// POUs/Motion/TF511x-KIN/03_DUTs/Trafo/KIN_STATICTRAFO_PARAM
{attribute 'hide'}
FUNCTION_BLOCK KIN_STATICTRAFO_PARAM
VAR_INPUT
	oid														:	UDINT := 0;
	TranslationX											:	LREAL := 0.0;
	TranslationY											:	LREAL := 0.0;
	TranslationZ											:	LREAL := 0.0;
                            								
	Rotation												: LREAL := 0.0;
	RotationAxis											: INT := 2;

END_VAR
VAR_OUTPUT

END_VAR
VAR
END_VAR

;

METHOD delete : BOOL
VAR_INPUT
END_VAR
	oid														:= 0;
	TranslationX											:= 0.0;
	TranslationY											:= 0.0;
	TranslationZ											:= 0.0;
                            								
	Rotation												:= 0.0;
	RotationAxis											:= 2;
delete	:= TRUE;
END_METHOD

END_FUNCTION_BLOCK

// POUs/Motion/TF511x-KIN/03_DUTs/Trafo/KIN_TOOLTRAFO_PARAM
{attribute 'hide'}
FUNCTION_BLOCK KIN_TOOLTRAFO_PARAM
VAR_INPUT
	oid														:	UDINT := 0;
	dx														: 	LREAL := 0.0;  (* Default Tooldata at WOS *)
	dy														: 	LREAL := 0.0;  (* Default Tooldata at WOS *)
	dz														:	LREAL := 0.0;  (* Default Tooldata at WOS *)

END_VAR
VAR_OUTPUT

END_VAR
VAR
END_VAR

;

METHOD delete : BOOL
VAR_INPUT
END_VAR
	oid														:= 0;
	dx														:= 0.0;  (* Default Tooldata at WOS *)
	dy														:= 0.0;  (* Default Tooldata at WOS *)
	dz														:= 0.0;  (* Default Tooldata at WOS *)
delete	:= TRUE;
END_METHOD

END_FUNCTION_BLOCK

// POUs/Motion/TF511x-KIN/KinChannel
FUNCTION_BLOCK KinChannel EXTENDS KIN_REF
VAR_INPUT
	Admin													:	KinAdmin;
END_VAR
VAR_OUTPUT
END_VAR
VAR
END_VAR

(* Kinematic Ctrl 										*)
(********************************************************)

(* work IO ********************************************************************)
(*	IO(); *)
	
(****************************************************************************)
(* Kinematic group control													*)
(****************************************************************************)
	Admin(
		ResetTrig			:= ,
		Enable			:= ,
		Override		:= ,
		ItpChannelId	:= ,
		AxesList		:= ,
		rKINRef			:= THIS^,
		Busy			=> ,
		Done			=> ,
		Error			=> ,
		ErrorId			=> );
(****************************************************************************)

END_FUNCTION_BLOCK

// POUs/Motion/VALUE_3D
{attribute 'no_check'}
FUNCTION_BLOCK VALUE_3D
VAR_INPUT                                                            
	Valid													:	BOOL ;
	X														:	LREAL;
	Y														:	LREAL;
	Z														:	LREAL;
END_VAR
VAR_OUTPUT
END_VAR
VAR
END_VAR

;

METHOD PUBLIC copy : BOOL //Return value = TRUE if execution finished
VAR_IN_OUT
	Source													:	VALUE_3D;
END_VAR
	Valid													:= Source.Valid;
	X														:= Source.X;
	Y														:= Source.Y;
	Z														:= Source.Z;
	copy													:= TRUE;
END_METHOD

METHOD PUBLIC delete : BOOL //Return value = TRUE if execution finished - Valid bit will not change
VAR_INPUT
END_VAR
	X					 									:= 0.0;	
	Y					 									:= 0.0;	
	Z					 									:= 0.0;	
	delete													:= TRUE;
END_METHOD

METHOD PUBLIC InPos : BOOL //Return value = TRUE axes is within window of checkPos values
VAR_IN_OUT
	CheckPos												:	VALUE_3D;
	Window													:	VALUE_3D;
END_VAR
InPos														:= CAM(CheckPos.X, X ,Window.X)
																AND CAM(CheckPos.Y, Y ,Window.Y)
																AND CAM(CheckPos.Z, Z ,Window.Z);
END_METHOD

METHOD PUBLIC InPosByAxisNo : BOOL //Return value = TRUE selected axis is within window of checkPos values
VAR_INPUT
	No					:	INT;
END_VAR
VAR_IN_OUT
	CheckPos			:	VALUE_3D;
	Window				:	VALUE_3D;
END_VAR
InPosByAxisNo													:= (CAM(CheckPos.X, X ,Window.X) OR No <> 1)
																AND (CAM(CheckPos.Y, Y ,Window.Y) OR No <> 2)
																AND (CAM(CheckPos.Z, Z ,Window.Z) OR No <> 3);
END_METHOD

METHOD PUBLIC InPosXY : BOOL //Return value = TRUE if axes are within window of checkPos values
VAR_IN_OUT
	CheckPos			:	VALUE_3D;
	Window				:	VALUE_3D;
END_VAR
InPosXY 													:= CAM(CheckPos.X, X ,Window.X)
																AND CAM(CheckPos.Y, Y ,Window.Y);
END_METHOD

METHOD PUBLIC InPosXZ : BOOL //Return value = TRUE if axes are within window of checkPos values
VAR_IN_OUT
	CheckPos			:	VALUE_3D;
	Window				:	VALUE_3D;
	
END_VAR
InPosXZ														:= CAM(CheckPos.X, X ,Window.X)
																AND CAM(CheckPos.Z, Z ,Window.Z);
END_METHOD

METHOD PUBLIC InPosYZ : BOOL //Return value = TRUE if axes are within window of checkPos values
VAR_IN_OUT
	CheckPos			:	VALUE_3D;
	Window				:	VALUE_3D;
	
END_VAR
InPosYZ													:= CAM(CheckPos.Y, Y ,Window.Y)
																AND CAM(CheckPos.Z, Z ,Window.Z);
END_METHOD

METHOD PUBLIC reset : BOOL //Delete data and reset valid , TRUE if execution finished
VAR_INPUT
END_VAR
Delete();
Valid														:= FALSE;
reset														:= TRUE;
END_METHOD

END_FUNCTION_BLOCK

// POUs/Motion/VALUE_6D
{attribute 'no_check'}
FUNCTION_BLOCK VALUE_6D 
VAR_INPUT
	Valid													:	BOOL ;
	X														:	LREAL;
	Y														:	LREAL;
	Z														:	LREAL;
	A														:		LREAL; //Rx
	B														:		LREAL; //Ry
	C														:		LREAL; //Rz	
END_VAR
VAR_OUTPUT
END_VAR
VAR
END_VAR

;

METHOD PUBLIC copy : BOOL //Return value = TRUE if execution finished
VAR_IN_OUT
	Source													:	VALUE_6D;
END_VAR
	Valid													:= Source.Valid;
	X														:= Source.X;
	Y														:= Source.Y;
	Z														:= Source.Z;
	A														:= Source.A;
	B														:= Source.B;
	C														:= Source.C;
	copy													:= TRUE;
END_METHOD

METHOD PUBLIC delete : BOOL //Return value = TRUE if execution finished - Valid bit will not change
VAR_INPUT
END_VAR
	X					 									:= 0.0;	
	Y					 									:= 0.0;	
	Z					 									:= 0.0;	
	A						 								:= 0.0;	
	B						 								:= 0.0;	
	C						 								:= 0.0;	
	delete													:= TRUE;
END_METHOD

METHOD PUBLIC inPos : BOOL //Return value = TRUE if axes are within window of checkPos values
VAR_IN_OUT
	CheckPos												:	VALUE_6D;
	Window													:	VALUE_6D;
END_VAR             										
VAR CONSTANT        										
END_VAR
InPos 														:= CAM(CheckPos.X, X, Window.X)
																AND CAM(CheckPos.Y, Y ,Window.Y)
																AND CAM(CheckPos.Z, Z,Window.Z)
																AND CAM(CheckPos.A, A, Window.A)
																AND CAM(CheckPos.B, B ,Window.B)
																AND CAM(CheckPos.C, C,Window.C);
END_METHOD

METHOD PUBLIC InPosABC : BOOL //Return value = TRUE if axes are within window of checkPos values
VAR_IN_OUT
	CheckPos												:	VALUE_6D;
	Window													:	VALUE_6D;
END_VAR                 									
VAR CONSTANT            									
END_VAR
InPosABC												 	:= CAM(CheckPos.A, A ,Window.A)
																AND CAM(CheckPos.B, B ,Window.B)
																AND CAM(CheckPos.C, C ,Window.C);
END_METHOD

METHOD PUBLIC InPosAC : BOOL //Return value = TRUE if axes are within window of checkPos values
VAR_IN_OUT
	CheckPos												:	VALUE_6D;
	Window													:	VALUE_6D;
END_VAR                 									
VAR CONSTANT            									
END_VAR
InPosAC													 	:= CAM(CheckPos.A, A ,Window.A)
																AND CAM(CheckPos.C, C ,Window.C);
END_METHOD

METHOD PUBLIC inPosByAxisNo : BOOL //Return value = TRUE selected axis is within window of checkPos values
VAR_INPUT
	No					:	INT;
END_VAR
VAR_IN_OUT
	CheckPos			:	VALUE_6D;
	Window				:	VALUE_6D;
END_VAR
inPosByAxisNo													:= (CAM(CheckPos.X, X ,Window.X) OR No <> 1)
																AND (CAM(CheckPos.Y, Y ,Window.Y) OR No <> 2)
																AND (CAM(CheckPos.Z, Z ,Window.Z) OR No <> 3)
																AND (CAM(CheckPos.A, A ,Window.A) OR No <> 4)
																AND (CAM(CheckPos.B, B ,Window.B) OR No <> 5)
																AND (CAM(CheckPos.C, C ,Window.C) OR No <> 6);
END_METHOD

METHOD PUBLIC inPosXY : BOOL //Return value = TRUE if axes are within window of checkPos values
VAR_IN_OUT
	CheckPos												:	VALUE_6D;
	Window													:	VALUE_6D;
END_VAR                 									
VAR CONSTANT            									
END_VAR
InPosXY													 	:= CAM(CheckPos.X, X ,Window.X)
																AND CAM(CheckPos.Y, Y ,Window.Y);
END_METHOD

METHOD PUBLIC InPosXYZ : BOOL //Return value = TRUE if axes are within window of checkPos values
VAR_IN_OUT
	CheckPos												:	VALUE_6D;
	Window													:	VALUE_6D;
END_VAR                 									
VAR CONSTANT            									
END_VAR
InPosXYZ												 	:= CAM(CheckPos.X, X ,Window.X)
																AND CAM(CheckPos.Y, Y ,Window.Y)
																AND CAM(CheckPos.Z, Z ,Window.Z);
END_METHOD

METHOD PUBLIC inPosXZ : BOOL //Return value = TRUE if axes are within window of checkPos values
VAR_IN_OUT
	CheckPos												:	VALUE_6D;
	Window													:	VALUE_6D;
END_VAR                 									
VAR CONSTANT            									
END_VAR
InPosXZ												 	:= CAM(CheckPos.X, X ,Window.X)
																AND CAM(CheckPos.Z, Z ,Window.Z);
END_METHOD

METHOD PUBLIC inPosYZ : BOOL //Return value = TRUE if axes are within window of checkPos values
VAR_IN_OUT
	CheckPos												:	VALUE_6D;
	Window													:	VALUE_6D;
END_VAR                 									
VAR CONSTANT            									
END_VAR
InPosYZ													 	:= CAM(CheckPos.Y, Y ,Window.Y)
																AND CAM(CheckPos.Z, Z ,Window.Z);
END_METHOD

METHOD PUBLIC reset : BOOL //Delete data and reset valid , TRUE if execution finished
VAR_INPUT
END_VAR
Delete(); 
Valid														:= FALSE;
reset														:= TRUE;
END_METHOD

END_FUNCTION_BLOCK

// POUs/Safety/Diag/SafetyIODeviceDiag_wEvents
{attribute 'no_check'}
FUNCTION_BLOCK SafetyIODeviceDiag_wEvents
VAR CONSTANT
	MIN_EVENT												:	INT := 1;
	MAX_EVENT												:	INT := 10;
	
//Event conn diag code xxxx					| FB1 - Msg 1..15
//Event conn diag code .4 					| FB2 - Msg 16
//Event conn diag code .5 					| FB3 - Msg 17
                                        	
//Event internal error 						| FB1 - Msg 18
                                        	
//Event send TextId 						| FB4 - Msg 19
                                        	
//Event send AX5xxx Err Chn 1 				| FB5 - Msg 20
//Event send AX5xxx Err Chn 1 				| FB6 - Msg 21
                                        	
//Event send Ex19 Err Debug 0x800E:0A 		| FB4 - Msg 22
//Event send Ex19 Err Debug 0x800E:0B		| FB5 - Msg 23
//Event send Ex19 Err Debug 0x800E:0C 		| FB6 - Msg 24
//Event send Ex19 Err Debug 0x800E:0D 		| FB7 - Msg 25
//Event send Ex19 Err Debug 0x800E:13 		| FB8 - Msg 26
//Event send Ex19 Err Debug 0x800E:14 		| FB9 - Msg 27
//Event send Ex19 Err Debug 0x800E:15		| FB10- Msg 28
                                        	
//Event send EL29 Err Debug 0x800E:0C 		| FB4 - Msg 30 (Querschluss bit 0..3)
//Event send EL29 Err Debug 0x800E:0C 		| FB4 - Msg 31 (Open load bit 4..7)
//Event send EL29 Err Debug 0x800E:0D		| FB5 - Msg 32
//Event send EL29 Err Debug 0x800E:0E 		| FB6 - Msg 33
//Event send EL29 Err Debug 0x800E:0E 		| FB7 - Msg 34
//Event send EL29 Err Debug 0x800E:0E 		| FB8 - Msg 35

                                        	
//Event send EK19 Err Debug 0x800E:0A		| FB4 - Msg 22 
//Event send EK19 Err Debug 0x800E:0B		| FB5 - Msg 23 
//Event send EK19 Err Debug 0x800E:0C 		| FB6 - Msg 24 
//Event send EK19 Err Debug 0x800E:0D 		| FB7 - Msg 25 
//Event send EK19 Err Debug 0x800E:0E	 	| FB8 - Msg 36..45
END_VAR
VAR_INPUT
	Enable													:	BOOL;	//FB will be processed as long as enable is TRUE 
	ConfirmTrig												:	BOOL;	//Resets error with rising edge 
	SourceId												:	UDINT;	//Multisource id 
	EcMasterDevId											:	UINT;	//Map to EtherCAT Master DevId
END_VAR                 									
VAR_OUTPUT              									
	Connected												:	BOOL;
	{attribute 'displaymode':='binary'}
	Status													:	DWORD;	//current status of event
	NoOfActiveEvents										:	INT;
END_VAR                 									

VAR(* internal *)
	state													:	INT := 0;
	{attribute 'displaymode':='binary'}
	ConnMsgDiagCode											:	BYTE;
	Read													:	SafetyIODeviceDiagRead;
   	Event													:	ARRAY [MIN_EVENT..MAX_EVENT] OF EventHandling; 
	DevTypeAndAddr											:	STRING(30);
    DebugData												:	 word;                 								                            	
	i														:	INT;
END_VAR

(* Safety IO device diag with events		V2	*)
(************************************************)

(* Status connected ***************************************************)
	Connected 												:= Read.AdsAddr.port <> 0;
	
(* Read adress and type ***********************************************)
	IF Enable AND Connected AND Read.MsgInfoDiag <> 0 OR State <> 0
	THEN
		CASE State OF
		0:	
			IF Read.MsgInfoDiag <> 0
			THEN
				Read(Execute := FALSE);
				Read(Execute := TRUE, EcMasterDevId := EcMasterDevId);
				State										:= State + 1;
			END_IF
			
		1: //Read diag data from device
			Read(Execute := TRUE, EcMasterDevId := EcMasterDevId);
			IF NOT Read.Busy
			THEN
	
				IF Read.Error
				THEN
					Event[1].Text1							:= SEL(Read.Name = '',Read.Name , '<ERR_READ_DIAG>');
					DevTypeAndAddr							:= SEL(Read.DevType = '', Read.DevType, '<Unknown>');
					DevTypeAndAddr							:= CONCAT(DevTypeAndAddr, CONCAT(' (Ec Addr.', CONCAT(TO_STRING(Read.AdsAddr.port),')')));	
					Event[1].Text2							:= CONCAT(' - ErrorID ', DWORD_TO_HEXSTR(TO_DWORD(Read.ErrorID),4,FALSE));
					Event[1].Text2							:= CONCAT(Event[1].Text2 , CONCAT(' in state ', TO_STRING(Read.DiagMsgTextId)));
					Event[1].SourceId						:= SourceId;
					Event[1].Flag							:= TRUE;
					State									:= 98;
				ELSIF Event[1].SourceId = 0
				THEN //Init device information 
					FOR i := MIN_EVENT TO MAX_EVENT
					DO
						Event[i].Text1						:= Read.Name;
						DevTypeAndAddr						:= CONCAT(Read.DevType, ' (FSOE Addr.');
						DevTypeAndAddr						:= CONCAT(DevTypeAndAddr, CONCAT(TO_STRING(Read.FSOEAddr), ')'));	
						Event[i].SourceId					:= SourceId;
					END_FOR
					State									:= 99;
				ELSE
					State									:= 99;
				END_IF		
				Read(Execute := FALSE);
			END_IF
			
		98: //Show internal error
			Event[1](
				Flag	:= Event[1].Flag AND NOT Event[1].ConfirmTrig,
				ConfirmTrig:= ConfirmTrig OR Read.MsgInfoDiag = 0, 
				MsgId	:= 18, 
				pText3	:= ADR(DevTypeAndAddr),
				Status	=> Status);	
			IF NOT Event[1].Status.31 
			THEN
				NoOfActiveEvents							:= 0;
				state										:= 0;
			ELSE
				NoOfActiveEvents							:= 1;
			END_IF
			
		99: //Fire events
			IF Read.MsgInfoDiag = 0 AND NOT Status.31
			THEN //Go back to 0 if messages cleared
				State 										:= 0;
			ELSE
				//Show connection error events
				_eventsConnDiag();
				
				//Fire device events
				IF Read.pDebugData <> 0 
				THEN //Safety devices without diag history object
					IF Read.DebugDataMaxId = 16#08 AND_THEN FIND(Read.DevType, 'AX580') <> 0
					THEN
						_eventsAX580x(Read.MsgInfoDiag <> 0);
					ELSIF Read.DebugDataMaxId = 16#10 AND_THEN Read.DevType = 'EL2904'
					THEN
						_eventsEL2904(Read.MsgInfoDiag <> 0);
					ELSIF Read.DebugDataMaxId = 16#40 AND_THEN Read.DevType = 'EK1914' 
					THEN
						_eventsEK1914(Read.MsgInfoDiag <> 0);
					ELSIF Read.DebugDataMaxId >= 16#10 
					THEN//EL1904 or EP1908
						_eventsEx190x(Read.MsgInfoDiag <> 0);		
					ELSE //Show internal error 
						Event[4](
							Flag	:= Read.MsgInfoDiag <> 0,
							ConfirmTrig:= ConfirmTrig OR Read.MsgInfoDiag = 0, 
							MsgId	:= 18, 
							Text2	:= CONCAT(' Invalid lenght of Coe object 0x800E for device ', TO_STRING(Read.DebugDataMaxId)),
							pText3	:= ADR(DevTypeAndAddr));	
					END_IF
				ELSE //TwinSAFE terminal with diag history  
					_eventsDiagHistory(Read.MsgInfoDiag <> 0);
				END_IF			
			END_IF		
						   	
			//Check whether one event is active **************************************
			NoOfActiveEvents 		 						:= 0;			
			Status											:= 0;						
			FOR i := MIN_EVENT TO MAX_EVENT
			DO 
				IF Event[i].Status.31 THEN NoOfActiveEvents := NoOfActiveEvents + 1 ; END_IF
				Status										:= Status OR Event[i].Status;
			END_FOR
		END_CASE
	END_IF

(*******************************************************************************)

METHOD PRIVATE _eventsAX580x : BOOL
VAR_INPUT
	ShowEvent										:	BOOL;
END_VAR
(* Fire AX5000 events ***********************************)
	//Send AX58xx diag code channel 1 
	IF Read.pDebugData^[1] = 0
	THEN
		Event[5].Text2										:= CONCAT('0x',DWORD_TO_HEXSTR(TO_DWORD(Read.pDebugData^[7]),4,FALSE));
	ELSE
		Event[5].Text2										:= '<Set CoE object 0xFA10:01 = 0>';
	END_IF
 
	Event[5](
		Flag	:= ShowEvent AND Read.msgSevyIsError ,
		ConfirmTrig:= ConfirmTrig, 
		MsgId	:= 20, 
		Class	:= ,
		pText3	:= ADR(DevTypeAndAddr));	
		
	//Send AX58xx diag code channel 2
	IF Read.pDebugData^[1] = 0
	THEN
		Event[6].Text2										:= CONCAT('0x',DWORD_TO_HEXSTR(TO_DWORD(Read.pDebugData^[8]),4,FALSE));
	ELSE
		Event[6].Text2										:=  '<Set CoE object 0xFA10:01 = 0>';
	END_IF
 
	Event[6](
		Flag	:= ShowEvent AND Read.msgSevyIsError ,
		ConfirmTrig:= ConfirmTrig, 
		MsgId	:= 21, 
		Class	:= ,
		pText3	:= ADR(Read.Name));

(******************************************************)
END_METHOD

METHOD PRIVATE _eventsConnDiag : BOOL
VAR_INPUT
END_VAR
(* Fire event for connection error code ************************************)
	ConnMsgDiagCode											:= 16#0F AND Read.MsgInfoDiag; 
	IF ConnMsgDiagCode <> 0 OR Event[1].Status.31
	THEN
		Event[1](
			Flag	:= ConnMsgDiagCode <> 0 AND NOT (ConnMsgDiagCode = 2#1101 AND Read.MsgInfoDiag.5),
			ConfirmTrig:= ConfirmTrig, 
			MsgId	:= ConnMsgDiagCode,  //1..15 		
			pText3	:= ADR(DevTypeAndAddr));	
	END_IF
	
	//Fire event xxx1 xxxx FSoE Slave error detected
	IF Read.MsgInfoDiag.4 OR Event[2].Status.31
	THEN
		Event[2](
			Flag	:= Read.MsgInfoDiag.4,
			ConfirmTrig:= ConfirmTrig, 
			MsgId	:= 16,		
			pText3	:= ADR(DevTypeAndAddr));	
	END_IF

(*
	//Fire event xx1x xxxx FSoE Slave notifies Failsafe Value active
	IF Read.MsgInfoDiag.5 OR Event[3].Status.31
	THEN
		Event[3](
			Flag	:= Read.MsgInfoDiag.5,
			ConfirmTrig:= ConfirmTrig, 
			MsgId	:= 17,		
			pText3	:= ADR(DevTypeAndAddr));		
	END_IF
*)	
	(*
	Tabelle 2-4: Diagnose-Informationen einer Connection
	Wert Beschreibung
	xxxx 0001 invalid command
	xxxx 0010 unknown command
	xxxx 0011 invalid connection ID
	xxxx 0100 invalid CRC
	xxxx 0101 Watchdog run out of time
	xxxx 0110 invalid FSoE-Adress
	xxxx 0111 invalid data
	xxxx 1000 invalid length of communicatoin parameter Kommunikationsparameterlänge
	xxxx 1001 invalid communicatoin parameter
	xxxx 1010 invalid operator parameter length
	xxxx 1011 invalid operator parameter
	xxxx 1100 FSoE Master Reset
	xxxx 1101 Module fault on slave detected with activated option "Modulfault is ComError"
	xxxx 1110 Module fault on EL290x at activated with option "Error achnowledge active"
	xxxx 1111 Slave not started or unexpected error argument
	
	*)
		
(***********************************************************************)
END_METHOD

METHOD PRIVATE _eventsDiagHistory : BOOL
VAR_INPUT
	ShowEvent										:	BOOL;
END_VAR
(* Send diag message textId ********************************************)
	Event[4](
		Flag	:= ShowEvent AND Read.msgSevyIsError ,
		ConfirmTrig:= ConfirmTrig, 
		MsgId	:= 19, 
		Text2	:= CONCAT('0x',DWORD_TO_HEXSTR(TO_DWORD(Read.DiagMsgTextId),4,FALSE)),
		pText3	:= ADR(DevTypeAndAddr));

(******************************************************)
END_METHOD

METHOD PRIVATE _eventsEK1914 : BOOL
VAR_INPUT
	ShowEvent										:	BOOL;
END_VAR
// Fire events for of EK1914 ****************************************)

		(* error during sensor-test *)
		Event[4].Flag 										:= Read.pDebugData^[16#0A] <> 0;
		IF Event[4].Flag OR Event[4].Status.31
		THEN
			DebugData										:= Read.pDebugData^[16#0A];
			Event[4].Text2									:= '';
			IF DebugData.0 THEN Event[4].Text2 				:= CONCAT(Event[4].Text2, '|1'); END_IF
			IF DebugData.1 THEN Event[4].Text2 				:= CONCAT(Event[4].Text2, '|2'); END_IF
		(*	IF DebugData.2 THEN Event[4].Text2 				:= CONCAT(Event[4].Text2, '|3'); END_IF
			IF DebugData.3 THEN Event[4].Text2 				:= CONCAT(Event[4].Text2, '|4');  END_IF
			IF DebugData.4 THEN Event[4].Text2 				:= CONCAT(Event[4].Text2, '|5'); END_IF
			IF DebugData.5 THEN Event[4].Text2 				:= CONCAT(Event[4].Text2, '|6'); END_IF
			IF DebugData.6 THEN Event[4].Text2 				:= CONCAT(Event[4].Text2, '|7'); END_IF
			IF DebugData.7 THEN Event[4].Text2 				:= CONCAT(Event[4].Text2, '|8');  END_IF *)
			Event[4].Text2 									:= CONCAT(Event[4].Text2, '|'); 			
			
			Event[4](
				Flag	:= ShowEvent ,
				ConfirmTrig:= ConfirmTrig, 
				MsgId	:= 22, 
				pText3	:= ADR(DevTypeAndAddr))	;
		END_IF

		(* Zweikanalauswertung fehlerhaft *)
		Event[5].Flag 										:= Read.pDebugData^[16#0B] <> 0;
		IF Event[5].Flag OR Event[5].Status.31
		THEN
			DebugData										:= Read.pDebugData^[16#0B];
			Event[5].Text2									:= '';
			IF DebugData.0 THEN Event[5].Text2 				:= CONCAT(Event[5].Text2, '|1+2'); END_IF
		(*	IF DebugData.1 THEN Event[5].Text2 				:= CONCAT(Event[5].Text2, '|3+4'); END_IF
			IF DebugData.2 THEN Event[5].Text2 				:= CONCAT(Event[5].Text2, '|5+6'); END_IF
			IF DebugData.3 THEN Event[5].Text2 				:= CONCAT(Event[5].Text2, '|7+8');  END_IF *)
			Event[5].Text2 									:= CONCAT(Event[5].Text2, '|'); 
			
			Event[5](
				Flag	:= ShowEvent ,
				ConfirmTrig:= ConfirmTrig, 
				MsgId	:= 23, 
				pText3	:= ADR(DevTypeAndAddr))	;
		END_IF

		(* Fehler Eingangspaar Trittmattenbetriebsart - Eingangspaar uneinig *)
		Event[6].Flag 										:= Read.pDebugData^[16#0C] <> 0;
		IF Event[6].Flag OR Event[6].Status.31
		THEN
			DebugData										:= Read.pDebugData^[16#0C];
			Event[6].Text2									:= '';
			IF DebugData.0 THEN Event[6].Text2 				:= CONCAT(Event[6].Text2, '|1+2'); END_IF
		(*	IF DebugData.1 THEN Event[6].Text2 				:= CONCAT(Event[6].Text2, '|3+4'); END_IF
			IF DebugData.2 THEN Event[6].Text2 				:= CONCAT(Event[6].Text2, '|5+6'); END_IF
			IF DebugData.3 THEN Event[6].Text2 				:= CONCAT(Event[6].Text2, '|7+8');  END_IF *)
			Event[6].Text2 									:= CONCAT(Event[6].Text2, '|'); 
			
			Event[6](
				Flag	:= ShowEvent ,
				ConfirmTrig:= ConfirmTrig, 
				MsgId	:= 24, 
				pText3	:= ADR(DevTypeAndAddr))	;
		END_IF

		(* Fehler Trittmattenbetriebsart Fremdeinspeisung *)
		Event[7].Flag 										:= Read.pDebugData^[16#0D] <> 0;
		IF Event[7].Flag OR Event[7].Status.31
		THEN
			DebugData										:= Read.pDebugData^[16#0D];
			Event[7].Text2									:= '';
			IF DebugData.0 THEN Event[7].Text2 				:= CONCAT(Event[7].Text2, '|1'); END_IF
			IF DebugData.1 THEN Event[7].Text2 				:= CONCAT(Event[7].Text2, '|2'); END_IF
		(*	IF DebugData.2 THEN Event[7].Text2 				:= CONCAT(Event[7].Text2, '|3'); END_IF
			IF DebugData.3 THEN Event[7].Text2 				:= CONCAT(Event[7].Text2, '|4');  END_IF
			IF DebugData.4 THEN Event[7].Text2 				:= CONCAT(Event[7].Text2, '|5'); END_IF
			IF DebugData.5 THEN Event[7].Text2 				:= CONCAT(Event[7].Text2, '|6'); END_IF
			IF DebugData.6 THEN Event[7].Text2 				:= CONCAT(Event[7].Text2, '|7'); END_IF
			IF DebugData.7 THEN Event[7].Text2 				:= CONCAT(Event[7].Text2, '|8');  END_IF *)
			Event[7].Text2 									:= CONCAT(Event[7].Text2, '|'); 
			
			Event[7](
				Flag	:= ShowEvent ,
				ConfirmTrig:= ConfirmTrig, 
				MsgId	:= 25, 
				pText3	:= ADR(DevTypeAndAddr))	;
		END_IF
		
		(* Fehler Ausgänge *)
		IF Read.pDebugData^[16#0E] <> 0 OR Event[8].Status.31 
		THEN
			DebugData										:= Read.pDebugData^[16#0E];
			
			CASE DebugData OF
			5:		Event[8].MsgId							:= 36;
			6:		Event[8].MsgId							:= 37;
			10:		Event[8].MsgId							:= 38;
			11:		Event[8].MsgId							:= 39;
			21..27:	Event[8].MsgId							:= 40;
			30..33:	Event[8].MsgId							:= 41;
			101:	Event[8].MsgId							:= 42;
			102:	Event[8].MsgId							:= 43;
			103:	Event[8].MsgId							:= 44;
			104:	Event[8].MsgId							:= 45;
			ELSE
				Event[8].MsgId								:= 0;
			END_CASE
				
			Event[8](
				Flag	:= ShowEvent AND Event[8].MsgId <> 0 ,
				ConfirmTrig:= ConfirmTrig, 
				MsgId	:= , 
				pText3	:= ADR(DevTypeAndAddr))	;
				
		END_IF		
(********************************************************************************)
END_METHOD

METHOD PRIVATE _eventsEL2904 : BOOL
VAR_INPUT
	ShowEvent										:	BOOL;
END_VAR
// Fire events for EL2904

	(* Fremeinspeisung oder Querschluss *)
	Event[4].Flag 										:= (Read.pDebugData^[16#0C] AND 16#000F) <> 0;
	IF Event[4].Flag OR Event[4].Status.31
	THEN
		DebugData										:= Read.pDebugData^[16#0C];
		Event[4].Text2									:= '';
		IF DebugData.0 THEN Event[4].Text2 				:= CONCAT(Event[4].Text2, '|1'); END_IF
		IF DebugData.1 THEN Event[4].Text2 				:= CONCAT(Event[4].Text2, '|2'); END_IF
		IF DebugData.2 THEN Event[4].Text2 				:= CONCAT(Event[4].Text2, '|3'); END_IF
		IF DebugData.3 THEN Event[4].Text2 				:= CONCAT(Event[4].Text2, '|4');  END_IF
		Event[4].Text2 									:= CONCAT(Event[4].Text2, '|'); 
			
		Event[4](
			Flag	:= ShowEvent ,
			ConfirmTrig:= ConfirmTrig, 
			MsgId	:= 30, 
			pText3	:= ADR(DevTypeAndAddr))	;
	END_IF

	(* Open load oder Mindeststrom (20mA) unterschritten, oder Maximalstrom ueberschritten (500mA) *)
	Event[5].Flag 										:= (Read.pDebugData^[16#0C] AND 16#00F0) <> 0;
	IF Event[5].Flag OR Event[5].Status.31
	THEN
		DebugData										:= Read.pDebugData^[16#0C];
		Event[5].Text2									:= '';
		IF DebugData.4 THEN Event[5].Text2 				:= CONCAT(Event[5].Text2, '|1'); END_IF
		IF DebugData.5 THEN Event[5].Text2 				:= CONCAT(Event[5].Text2, '|2'); END_IF
		IF DebugData.6 THEN Event[5].Text2 				:= CONCAT(Event[5].Text2, '|3'); END_IF
		IF DebugData.7 THEN Event[5].Text2 				:= CONCAT(Event[5].Text2, '|4');  END_IF
		Event[5].Text2 									:= CONCAT(Event[5].Text2, '|'); 
		
		Event[5](
			Flag	:= ShowEvent ,
			ConfirmTrig:= ConfirmTrig, 
			MsgId	:= 31, 
			pText3	:= ADR(DevTypeAndAddr));	
	END_IF
	
	(* Fehler Feldspannung Power Kontakte *)
	Event[6].Flag 										:= Read.pDebugData^[16#0D] <> 0;
	IF Event[6].Flag OR Event[6].Status.31
	THEN
		DebugData										:= Read.pDebugData^[16#0D];
		Event[6].Text2									:= '';
		IF DebugData.0 THEN 
			Event[6].Text2 								:= CONCAT(Event[6].Text2, '|Y'); 
		ELSE                                                                       
			Event[6].Text2 								:= CONCAT(Event[6].Text2, '|N'); 
		END_IF                                                                     
		IF DebugData.1 THEN                                                        
			Event[6].Text2 								:= CONCAT(Event[6].Text2, '|Y'); 
		ELSE                                                                       
			Event[6].Text2 								:= CONCAT(Event[6].Text2, '|N'); 
		END_IF
		Event[6].Text2 									:= CONCAT(Event[6].Text2, '|'); 
		
		Event[6](
			Flag	:= ShowEvent ,
			ConfirmTrig:= ConfirmTrig, 
			MsgId	:= 32, 
			pText3	:= ADR(DevTypeAndAddr))	;
	END_IF
	
	(* Temperaturfehler *)
	IF Read.pDebugData^[16#0E] <> 0 OR Event[7].Status.31 OR Event[8].Status.31 OR Event[9].Status.31
	THEN
		DebugData										:= Read.pDebugData^[16#0E];
		
		//Uebertemperatur
		Event[7](
			Flag	:= ShowEvent AND(DebugData.0 OR DebugData.1 OR DebugData.2),
			ConfirmTrig:= ConfirmTrig, 
			MsgId	:= 33, 
			pText3	:= ADR(DevTypeAndAddr));	
			
		//Untertemperatur
		Event[8](
			Flag	:= ShowEvent AND(DebugData.3 OR DebugData.4 OR DebugData.5),
			ConfirmTrig:= ConfirmTrig, 
			MsgId	:= 34, 
			pText3	:= ADR(DevTypeAndAddr))	;
			
		//Temp. Differenz
		Event[9](
			Flag	:= ShowEvent AND(DebugData.6 OR DebugData.6),
			ConfirmTrig:= ConfirmTrig, 
			MsgId	:= 35, 
			pText3	:= ADR(DevTypeAndAddr))	;
	END_IF
		
(***********************************************************************)
END_METHOD

METHOD PRIVATE _eventsEx190x : BOOL
VAR_INPUT
	ShowEvent										:	BOOL;
END_VAR
VAR
	DebugData												:	WORD;
END_VAR
// Fire events for EL1904 and EP1908 errors

	(* error during sensor-test *)
	Event[4].Flag 										:= Read.pDebugData^[16#0A] <> 0;
	IF Event[4].Flag OR Event[4].Status.31
	THEN
		DebugData										:= Read.pDebugData^[16#0A];
		Event[4].Text2									:= '';
		IF DebugData.0 THEN Event[4].Text2 				:= CONCAT(Event[4].Text2, '|1'); END_IF
		IF DebugData.1 THEN Event[4].Text2 				:= CONCAT(Event[4].Text2, '|2'); END_IF
		IF DebugData.2 THEN Event[4].Text2 				:= CONCAT(Event[4].Text2, '|3'); END_IF
		IF DebugData.3 THEN Event[4].Text2 				:= CONCAT(Event[4].Text2, '|4');  END_IF
		IF DebugData.4 THEN Event[4].Text2 				:= CONCAT(Event[4].Text2, '|5'); END_IF
		IF DebugData.5 THEN Event[4].Text2 				:= CONCAT(Event[4].Text2, '|6'); END_IF
		IF DebugData.6 THEN Event[4].Text2 				:= CONCAT(Event[4].Text2, '|7'); END_IF
		IF DebugData.7 THEN Event[4].Text2 				:= CONCAT(Event[4].Text2, '|8');  END_IF
		Event[4].Text2 									:= CONCAT(Event[4].Text2, '|'); 
		
		Event[4](
			Flag	:= ShowEvent ,
			ConfirmTrig:= ConfirmTrig, 
			MsgId	:= 22, 
			pText3	:= ADR(DevTypeAndAddr))	;
	END_IF

	(* Zweikanalauswertung fehlerhaft *)
	Event[5].Flag 										:= Read.pDebugData^[16#0B] <> 0;
	IF Event[5].Flag OR Event[5].Status.31
	THEN
		DebugData										:= Read.pDebugData^[16#0B];
		Event[5].Text2									:= '';
		IF DebugData.0 THEN Event[5].Text2 				:= CONCAT(Event[5].Text2, '|1+2'); END_IF
		IF DebugData.1 THEN Event[5].Text2 				:= CONCAT(Event[5].Text2, '|3+4'); END_IF
		IF DebugData.2 THEN Event[5].Text2 				:= CONCAT(Event[5].Text2, '|5+6'); END_IF
		IF DebugData.3 THEN Event[5].Text2 				:= CONCAT(Event[5].Text2, '|7+8');  END_IF
		Event[5].Text2 									:= CONCAT(Event[5].Text2, '|'); 		
	
		Event[5](
			Flag	:= ShowEvent ,
			ConfirmTrig:= ConfirmTrig, 
			MsgId	:= 23, 
			pText3	:= ADR(DevTypeAndAddr))	;
	END_IF

	(* Fehler Eingangspaar Trittmattenbetriebsart - Eingangspaar uneinig *)
	Event[6].Flag 										:= Read.pDebugData^[16#0C] <> 0;
	IF Event[6].Flag OR Event[6].Status.31
	THEN
		DebugData										:= Read.pDebugData^[16#0C];
		Event[6].Text2									:= '';
		IF DebugData.0 THEN Event[6].Text2 				:= CONCAT(Event[6].Text2, '|1+2'); END_IF
		IF DebugData.1 THEN Event[6].Text2 				:= CONCAT(Event[6].Text2, '|3+4'); END_IF
		IF DebugData.2 THEN Event[6].Text2 				:= CONCAT(Event[6].Text2, '|5+6'); END_IF
		IF DebugData.3 THEN Event[6].Text2 				:= CONCAT(Event[6].Text2, '|7+8');  END_IF
		Event[6].Text2 									:= CONCAT(Event[6].Text2, '|'); 
				
		Event[6](
			Flag	:= ShowEvent ,
			ConfirmTrig:= ConfirmTrig, 
			MsgId	:= 24, 
			pText3	:= ADR(DevTypeAndAddr))	;
	END_IF

	(* Fehler Trittmattenbetriebsart Fremdeinspeisung *)
	Event[7].Flag 										:= Read.pDebugData^[16#0D] <> 0;
	IF Event[7].Flag OR Event[7].Status.31
	THEN
		DebugData										:= Read.pDebugData^[16#0D];
		Event[7].Text2									:= '';
		IF DebugData.0 THEN Event[7].Text2 				:= CONCAT(Event[7].Text2, '|1'); END_IF
		IF DebugData.1 THEN Event[7].Text2 				:= CONCAT(Event[7].Text2, '|2'); END_IF
		IF DebugData.2 THEN Event[7].Text2 				:= CONCAT(Event[7].Text2, '|3'); END_IF
		IF DebugData.3 THEN Event[7].Text2 				:= CONCAT(Event[7].Text2, '|4');  END_IF
		IF DebugData.4 THEN Event[7].Text2 				:= CONCAT(Event[7].Text2, '|5'); END_IF
		IF DebugData.5 THEN Event[7].Text2 				:= CONCAT(Event[7].Text2, '|6'); END_IF
		IF DebugData.6 THEN Event[7].Text2 				:= CONCAT(Event[7].Text2, '|7'); END_IF
		IF DebugData.7 THEN Event[7].Text2 				:= CONCAT(Event[7].Text2, '|8');  END_IF
		Event[7].Text2 									:= CONCAT(Event[7].Text2, '|'); 
		
		Event[7](
			Flag	:= ShowEvent ,
			ConfirmTrig:= ConfirmTrig, 
			MsgId	:= 25, 
			pText3	:= ADR(DevTypeAndAddr))	;
	END_IF
	

//Events for EP1908 ****************************************************************)
IF Read.DebugDataMaxId > 16#10 THEN

	(* Fehler der Drehzahlueberwachung:Ueberdrehzahl *)
	Event[8].Flag 										:= Read.pDebugData^[16#13] <> 0;
	IF Event[8].Flag OR Event[8].Status.31
	THEN
		DebugData										:= Read.pDebugData^[16#13];
		Event[8].Text2									:= '';
		IF DebugData.0 THEN Event[8].Text2 				:= CONCAT(Event[8].Text2, '|1'); END_IF
		IF DebugData.1 THEN Event[8].Text2 				:= CONCAT(Event[8].Text2, '|2'); END_IF
		IF DebugData.2 THEN Event[8].Text2 				:= CONCAT(Event[8].Text2, '|3'); END_IF
		IF DebugData.3 THEN Event[8].Text2 				:= CONCAT(Event[8].Text2, '|4');  END_IF
		IF DebugData.4 THEN Event[8].Text2 				:= CONCAT(Event[8].Text2, '|5'); END_IF
		IF DebugData.5 THEN Event[8].Text2 				:= CONCAT(Event[8].Text2, '|6'); END_IF
		IF DebugData.6 THEN Event[8].Text2 				:= CONCAT(Event[8].Text2, '|7'); END_IF
		IF DebugData.7 THEN Event[8].Text2 				:= CONCAT(Event[8].Text2, '|8');  END_IF
		Event[8].Text2 									:= CONCAT(Event[8].Text2, '|'); 
		
		Event[8](
			Flag	:= ShowEvent ,
			ConfirmTrig:= ConfirmTrig, 
			MsgId	:= 26, 
			pText3	:= ADR(DevTypeAndAddr))	;
	END_IF
	
	(* Fehler in der Betriebsart: Two Channel Sync Velocity *)
	Event[9].Flag 										:= Read.pDebugData^[16#14] <> 0;
	IF Event[9].Flag OR Event[9].Status.31
	THEN
		DebugData										:= Read.pDebugData^[16#14];
		Event[9].Text2									:= '';
		IF DebugData.0 THEN Event[9].Text2 				:= CONCAT(Event[9].Text2, '|1+2'); END_IF
		IF DebugData.1 THEN Event[9].Text2 				:= CONCAT(Event[9].Text2, '|3+4'); END_IF
		IF DebugData.2 THEN Event[9].Text2 				:= CONCAT(Event[9].Text2, '|5+6'); END_IF
		IF DebugData.3 THEN Event[9].Text2 				:= CONCAT(Event[9].Text2, '|7+8');  END_IF
		Event[9].Text2 									:= CONCAT(Event[9].Text2, '|'); 
		
		Event[9](
			Flag	:= ShowEvent ,
			ConfirmTrig:= ConfirmTrig, 
			MsgId	:= 27, 
			pText3	:= ADR(DevTypeAndAddr))	;
	END_IF
	
	(* Fehler in der Betriebsart: Two Channel Sync Velocity UND Two Channel Encoder Velocity Control*)
	Event[10].Flag 										:= Read.pDebugData^[16#15] <> 0;
	IF Event[10].Flag OR Event[10].Status.31
	THEN
		DebugData										:= Read.pDebugData^[16#15];
		Event[10].Text2									:= '';
		IF DebugData.0 THEN Event[10].Text2 			:= CONCAT(Event[10].Text2, '|1+2'); END_IF
		IF DebugData.1 THEN Event[10].Text2 			:= CONCAT(Event[10].Text2, '|3+4'); END_IF
		IF DebugData.2 THEN Event[10].Text2 			:= CONCAT(Event[10].Text2, '|5+6'); END_IF
		IF DebugData.3 THEN Event[10].Text2 			:= CONCAT(Event[10].Text2, '|7+8');  END_IF
		Event[10].Text2 								:= CONCAT(Event[10].Text2, '|'); 
		
		Event[10](
			Flag	:= ShowEvent ,
			ConfirmTrig:= ConfirmTrig, 
			MsgId	:= 28, 
			pText3	:= ADR(DevTypeAndAddr))	;
	END_IF
END_IF

(************************************************************************************)
END_METHOD

END_FUNCTION_BLOCK

// POUs/Safety/Diag/SafetyIODeviceDiagRead
{attribute 'no_check'}
{attribute 'enable_dynamic_creation'}
FUNCTION_BLOCK SafetyIODeviceDiagRead EXTENDS FbBase
VAR CONSTANT
	bitTwinSAFETerm											:	BYTE := 0; //Ex1918,ELx9xx, etc. (2nd generation of TwinSAFE devices with CoE Index 10F3 Diag History included)
	bitSafetyTerm											:	BYTE := 1; //EL1904,EL2904,EK1914,EP1908 (Diagnoses provided via CoE Index 0x800E FSOE Internal Data, Debug 1..x) 
 	bitAX58xx												:	BYTE := 2; //AX5805,AX5806 (Diag via CoE index 0xFA10)
END_VAR
VAR_INPUT
	EcMasterDevId											:	UINT;	//EtherCAT Master DevId
END_VAR                 									
VAR_OUTPUT              									 
	AdsAddr											AT %I*	:	AMSADDR; //Link to terminal/box/device AMS Net Addr.
	{attribute 'displaymode':='binary'}
	MsgInfoDiag										AT %I*	:	USINT; 	//Link to connection messagediag of EL69xx (Needs to be enabled for alias of device)
//	{attribute 'displaymode':='hexadecimal'}
//	MsgInfoState									AT %I*	:	USINT; 	//Link to connection message state of EL69xx (Needs to be enabled for alias of device)	
	DevType													:	STRING(15); //CoE index 1008 / e.g. EL1908, EP1957-0022, etc...
	Name													:	STRING(31);	//Device name as defined in system manager configuration								
	FSOEAddr												:	WORD; //CoE index 0xF980
	DiagMsgSeverity											:	UINT; //Info (0) Warning (1) or Error (2)
	{attribute 'displaymode':='hexadecimal'}
	DiagMsgTextId											: 	UINT; //CoE Index 10F3 newest diagnoses message TextID (xyzz -> X =Type | y = Source | zz = Message ID)
	{attribute 'displaymode':='hexadecimal'}
	pDebugData												:	POINTER TO ARRAY[0..64] OF WORD; //Pointer to CoE index 0x800E - FSOE Internal Data - Debug 1-x for diag of "Safety Terminals" (or CoE Index 0xFA10 for AX58xx)
	DebugDataMaxId											:	UINT; //Max index for pointer pDebugData to array of word (Debug 1..x) if 0 data are invalid		
END_VAR                 									

VAR(* internal *)    
	{attribute 'displaymode':='bin'}
	DevCategory												:	BYTE;
	IOF_GetBoxNameByAddr									:	IOF_GetBoxNameByAddr := (TMOUT	:= DEFAULT_ADS_TIMEOUT);
	EcCoEReadDiagMsg										:	EcCoEReadNewestDiagMsg ;              									
	EcCoESdoReadEx											:	FB_EcCoESdoReadEx := (tTimeout := DEFAULT_ADS_TIMEOUT);       
	i														:	INT;  								                            	
END_VAR
(*
Tabelle 2-4: Diagnose-Informationen einer Connection
Wert Beschreibung
xxxx 0001 invalid command
xxxx 0010 unknown command
xxxx 0011 invalid connection ID
xxxx 0100 invalid CRC
xxxx 0101 Watchdog run out of time
xxxx 0110 invalid FSoE-Adress
xxxx 0111 invalid data
xxxx 1000 invalid length of communicatoin parameter Kommunikationsparameterlänge
xxxx 1001 invalid communicatoin parameter
xxxx 1010 invalid operator parameter length
xxxx 1011 invalid operator parameter
xxxx 1100 FSoE Master Reset
xxxx 1101 Module fault on slave detected with activated option "Modulfault is ComError"
xxxx 1110 Module fault on EL290x at activated with option "Error achnowledge active"
xxxx 1111 Slave not started or unexpected error argument

xxx1 xxxx FSoE Slave error detected
xx1x xxxx FSoE Slave notifies Failsafe Value active
x1xx xxxx StartUp
1xxx xxxx FSoE Master notifies Failsafe Value active
*)

(* IO Safety Terminal Status Diag		V2.0	*)
(************************************************)

(* Trigger to read diag **********************************************)
	rtExecute(CLK := Execute);
	
(* Read adress and type ***********************************************)
	CASE state OF
	0:
		Busy 												:= FALSE;
		IF NOT Execute
		THEN
			Done											:= FALSE;
			Error											:= FALSE;
			ErrorId											:= 0;					
		END_IF
		
		IF rtExecute.Q
		THEN
			Busy 											:= TRUE;
			Done											:= FALSE;
			Error											:= FALSE;
			ErrorId											:= 0;
			DiagMsgTextId									:= 0;
			DiagMsgSeverity									:= 0;

			EcCoESdoReadEx(bExecute := FALSE, bCompleteAccess := FALSE);
			IOF_GetBoxNameByAddr(Start := FALSE);
			EcCoEReadDiagMsg(Execute := FALSE);
			
			IF DevCategory.bitTwinSAFETerm
			THEN
				state 										:= 10;	
			ELSIF DevCategory.bitSafetyTerm
			THEN
				state 										:= SEL(DebugDataMaxId = 0, 21, 20);
			ELSIF DevCategory.bitAX58xx				
			THEN 
				state 										:= 30;
				
			ELSE //Read more device information 
				state										:= state + 1;				
			END_IF
		
		END_IF

	1: (* read FSOE adress *)
		EcCoESdoReadEx(
			sNetId			:= F_CreateAmsNetId(nIds := AdsAddr.netId ),
			nSlaveAddr		:= AdsAddr.port,
			nSubIndex		:= 16#1,
			nIndex			:= 16#F980,
			pDstBuf			:= ADR(FSOEAddr),
			cbBufLen		:= SIZEOF(FSOEAddr),
			bExecute		:= TRUE,
			tTimeout		:=  (* Default *),
			bCompleteAccess	:= ,
			bBusy			=> ,
			bError			=> ,
			nErrId			=> );
			
		IF NOT EcCoESdoReadEx.bBusy
		THEN
			IF EcCoESdoReadEx.bError 
			THEN
				Busy 										:= FALSE;
				Error										:= TRUE;
				ErrorId										:= EcCoESdoReadEx.nErrId;
				DiagMsgTextId								:= TO_UINT(state);
				state										:= 0;
			ELSE      									
				state 										:= state + 1;
			END_IF
			EcCoESdoReadEx(bExecute := FALSE);
		END_IF

	2: //Ready name from system manager configuration
		IOF_GetBoxNameByAddr(
			NETID		:='' , (* Local *)
			DEVICEID	:= UINT_TO_UDINT(EcMasterDevId) ,
			BOXADDR		:= AdsAddr.port ,
			START		:= EcMasterDevId <> 0,
			BOXNAME		=> );
			
		IF NOT IOF_GetBoxNameByAddr.Busy
		THEN
			IF IOF_GetBoxNameByAddr.Err 
			THEN
				Busy 										:= FALSE;
				Error										:= TRUE;
				ErrorId										:= IOF_GetBoxNameByAddr.ERRID;
				DiagMsgTextId								:= TO_UINT(state);
				state										:= 0;
			ELSIF IOF_GetBoxNameByAddr.Start
			THEN
				state 										:= state + 1;
			ELSE //No box name to read
				Name										:= CONCAT('EtherCAT Addr.',TO_STRING(AdsAddr.port));
			END_IF
			IOF_GetBoxNameByAddr(START := FALSE);
		END_IF
		
	3:  (* read device name e.g. EL1904 *)
		EcCoESdoReadEx(bExecute	:= TRUE, nIndex	:= 16#1008, nSubIndex := 16#0, pDstBuf := ADR(DevType),cbBufLen	:= SIZEOF(DevType));

		IF NOT EcCoESdoReadEx.bBusy
		THEN
			IF EcCoESdoReadEx.bError 
			THEN
				Busy 										:= FALSE;
				Error										:= TRUE;
				ErrorId										:= EcCoESdoReadEx.nErrId;
				DiagMsgTextId								:= TO_UINT(state);
				state										:= 0;
			ELSE       
				 //Delte type from name if in brakets 
				Name										:= DELETE(IOF_GetBoxNameByAddr.BOXNAME, LEN(DevType) + 2 , FIND(IOF_GetBoxNameByAddr.BOXNAME,DevType) - 1);
                             	
				IF DevType = 'AX5806' OR_ELSE DevType = 'AX5805'
				THEN
					DevCategory.bitAX58xx					:= TRUE;
					state 									:= 30;
				ELSIF DevType = 'EL1904' OR_ELSE DevType = 'EL2904' OR_ELSE DevType = 'EK1914' OR_ELSE DevType = 'EP1908'
				THEN
					DevCategory.bitSafetyTerm 				:= TRUE;
					state 									:= SEL(DebugDataMaxId = 0, 21, 20);
				ELSE
					DevCategory.bitTwinSAFETerm				:= TRUE;
					state 									:= 10;
				END_IF
				
			END_IF
			EcCoESdoReadEx(bExecute := FALSE);
		END_IF

	(* Read diagnoses latest entry from diag history ***********************************)	
	10: 
		EcCoEReadDiagMsg(Execute := TRUE, AdsAddr := AdsAddr);
		IF NOT EcCoEReadDiagMsg.Busy
		THEN
			IF EcCoEReadDiagMsg.Error 
			THEN
				Busy 										:= FALSE;
				Error										:= TRUE;
				ErrorId										:= EcCoEReadDiagMsg.ErrorID;
				DiagMsgTextId								:= TO_UINT(state);
				state										:= 0;				
			ELSE
				DiagMsgTextId								:= EcCoEReadDiagMsg.MsgId;
				DiagMsgSeverity								:= EcCoEReadDiagMsg.MsgSeverity;
				Done										:= TRUE;
				Busy										:= FALSE;
				State										:= 0;
			END_IF
		END_IF
		
	(* Read lenght of 0x800E:0 FSOE internal data.Debug terminal *********************************)
	20:
		EcCoESdoReadEx(bExecute	:= DebugDataMaxId = 0, nIndex	:= 16#800E, nSubIndex := 16#0, pDstBuf := ADR(DebugDataMaxId),cbBufLen	:= SIZEOF(DebugDataMaxId));

		IF NOT EcCoESdoReadEx.bBusy
		THEN
			IF EcCoESdoReadEx.bError 
			THEN
				Busy 										:= FALSE;
				Error										:= TRUE;
				ErrorId										:= EcCoESdoReadEx.nErrId;
				DiagMsgTextId								:= TO_UINT(state);
				state										:= 0;
			ELSIF DebugDataMaxId = 0
			THEN
				Busy 										:= FALSE;
				Error										:= TRUE;
				ErrorId										:= E_AdsErr.DEVICE_INVALIDPARM; //Lenght of index cannot be 0
				DiagMsgTextId								:= TO_UINT(state);
				state										:= 0;				
			ELSIF pDebugData = 0
			THEN                                  	
				pDebugData									:= __NEW(WORD,TO_UDINT(DebugDataMaxId + 1)); //e.g. 16 words = 32 bytes + 1 word for index 0 (which is in fact a byte  				
				IF PARAM.ENABLE_DEBUG_MSG_DYNAMIC_MEM_ALLOCATION
				THEN
					AdsLogHint('EngineeringToolbox | FB SafetyIOReadDiag | An instance allocated %s bytes from the dynamic memory of the ADS router memory pool', TO_STRING((DebugDataMaxId * 2) + 2));
				END_IF
				state 										:= state + 1;
			ELSE
				state 										:= state + 1;
			END_IF
			EcCoESdoReadEx(bExecute := FALSE);
		END_IF	
		
	21://Read all debug data from terminal
		EcCoESdoReadEx(bExecute	:= TRUE, nIndex	:= 16#800E, nSubIndex := 16#0, pDstBuf := pDebugData ,cbBufLen := TO_UDINT(DebugDataMaxId * 2) + SIZEOF(DebugDataMaxId) , bCompleteAccess := TRUE);

		IF NOT EcCoESdoReadEx.bBusy
		THEN
			IF EcCoESdoReadEx.bError 
			THEN
				IF pDebugData = 0
				THEN
					DebugDataMaxId							:= 0;
				END_IF
				Busy 										:= FALSE;
				Error										:= TRUE;
				ErrorId										:= EcCoESdoReadEx.nErrId;
				DiagMsgTextId								:= TO_UINT(state);
				state										:= 0;
			ELSE                                    		
				Done										:= TRUE;
				Busy										:= FALSE;
				DiagMsgSeverity								:= 2;
				State										:= 0;					
			END_IF
			EcCoESdoReadEx(bExecute := FALSE, bCompleteAccess := FALSE );
		END_IF			
	
	(* Read diag data from AX58xx *********************************)
	30:
		IF pDebugData = 0
		THEN
			DebugDataMaxId									:= 16#8;
			pDebugData										:= __NEW(WORD,TO_UDINT(DebugDataMaxId + 1));
			
			IF PARAM.ENABLE_DEBUG_MSG_DYNAMIC_MEM_ALLOCATION
			THEN
				AdsLogHint('EngineeringToolbox | FB SafetyIOReadDiag | An instance allocated %s bytes from the dynamic memory of the ADS router memory pool', '18');
			END_IF				
		END_IF
		
		EcCoESdoReadEx(bExecute	:= TRUE, nIndex	:= 16#FA10, nSubIndex := 16#0, pDstBuf := pDebugData, cbBufLen	:= TO_UDINT(DebugDataMaxId * 2) + SIZEOF(DebugDataMaxId),bCompleteAccess := TRUE);

		IF NOT EcCoESdoReadEx.bBusy
		THEN
			IF EcCoESdoReadEx.bError 
			THEN
				IF pDebugData = 0
				THEN
					DebugDataMaxId							:= 0;
				END_IF
				Busy 										:= FALSE;
				Error										:= TRUE;
				ErrorId										:= EcCoESdoReadEx.nErrId;
				DiagMsgTextId								:= TO_UINT(state);
				state										:= 0;
			ELSE                                    		
				Done										:= TRUE;
				Busy										:= FALSE;
				DiagMsgSeverity								:= 2;
				State										:= 0;	
			END_IF
			EcCoESdoReadEx(bExecute := FALSE, bCompleteAccess := FALSE);
		END_IF	
	ELSE
		;
	END_CASE
			
(*********************************************************************************************)

METHOD FB_exit : BOOL
VAR_INPUT
	bInCopyCode : BOOL; // if TRUE, the exit method is called for exiting an instance that is copied afterwards (online change).
END_VAR
IF NOT bInCopyCode AND pDebugData <> 0
THEN //Release memory in case the PLC stopps
	__DELETE(pDebugData);
	DebugDataMaxId								:= 0;
END_IF
END_METHOD

{attribute 'monitoring' := 'call'}
PROPERTY PUBLIC msgSevyIsError : BOOL
GET
msgSevyIsError := DiagMsgSeverity = 2;
END_GET
END_PROPERTY

{attribute 'monitoring' := 'call'}
PROPERTY PUBLIC msgSevyIsInfo : BOOL
GET
msgSevyIsInfo := DiagMsgSeverity = 0;
END_GET
END_PROPERTY

{attribute 'monitoring' := 'call'}
PROPERTY PUBLIC msgSevyIsWarning : BOOL
GET
msgSevyIsWarning := DiagMsgSeverity = 1;
END_GET
END_PROPERTY

END_FUNCTION_BLOCK

// POUs/Safety/Diag/SafetyIOsDiag
{attribute 'no_check'}
FUNCTION_BLOCK SafetyIOsDiag
VAR CONSTANT
	MIN_TERM												:	INT := 1;
	MAX_TERM												:	INT := PARAM.SAFETY_IO_TERM_DIAG_MAX;
END_VAR                     								
VAR_INPUT                   								
	Enable													:	BOOL;	//FB will be processed as long as enable is TRUE 
	ConfirmTrig												:	BOOL;	//Resets error with rising edge 
	SourceMultiId											:	UDINT := 100310;
	EcMasterDevId											:	UINT;	//Map to EtherCAT Master DevId
END_VAR                     								
VAR_OUTPUT                  	
	{attribute 'displaymode':='binary'}
	Status													:	DWORD;	//Current status of all events
	NoOfActiveEvents										:	INT;
END_VAR
VAR (* Events/Blocks/Var internal *)
	DevNo													:	ARRAY [MIN_TERM..MAX_TERM] OF SafetyIODeviceDiag_wEvents;
    tonStartupDelay											:	ton := (PT := T#200MS);                 								
	i														:	INT := MIN_TERM;
	StartCnt												:	BYTE := 0;
                           	
END_VAR

(* EL Safety IO Terminal Diag							*)
(********************************************************)

(* start one after the other ***************************)
	IF StartCnt < MAX_TERM 
	THEN
		tonStartupDelay(IN := TRUE);
		IF tonStartupDelay.Q
		THEN
			tonStartupDelay(IN := FALSE);
			StartCnt 										:= StartCnt + 1;
			DevNo[StartCnt].SourceId						:= SourceMultiId + StartCnt;
			DevNo[StartCnt].EcMasterDevId					:= EcMasterDevId;
			
		END_IF
	END_IF

(* terminal event ***************************************)
	Status 													:= 0;
	NoOfActiveEvents										:= 0;
	FOR i := MIN_TERM TO MAX_TERM
	DO
		DevNo[i](
			Enable			:= Enable AND StartCnt >= i,
			ConfirmTrig		:= ConfirmTrig,
			SourceId		:= ,
			EcMasterDevId	:= ,
			Status			=> );
				
		IF DevNo[i].Connected
		THEN
			IF DevNo[i].Status.31 THEN NoOfActiveEvents := NoOfActiveEvents + DevNo[i].NoOfActiveEvents ; END_IF
			Status											:= Status OR DevNo[i].Status;
		ELSE
			EXIT; 
		END_IF
	END_FOR

(*******************************************************)

END_FUNCTION_BLOCK

// POUs/Safety/Diag/SafetyLogicTerminalDiag
{attribute 'no_check'}
FUNCTION_BLOCK SafetyLogicTerminalDiag // EL6910, EL and EP devices with integrated TwinSAFE logic 
VAR CONSTANT
	MIN_FB													:	INT := 1;
	MAX_FB													:	INT := PARAM.SAFETY_PLC_TERM_DIAG_MAX_FB;
	
	TIMEOUT_CYCLE_COUNTER									:	TIME := T#1S;
	DEFAULT_SOURCE_ID										:	UDINT := 100300; //Multisource id 
	INVALID_SAFETY_LOGIC_STATE								:	USINT := 255;
END_VAR                 									
VAR_INPUT               									
	Enable													:	BOOL := TRUE;	//FB will be processed as long as enable is TRUE 
	Quit													:	BOOL;			//Resets error with rising edge 
	IO														:	Eyx9xx;			
END_VAR
VAR_OUTPUT
	{attribute 'displaymode':='binary'}
	Status													:	DWORD; 			//current sttus of all events
	NoOfActiveEvents										:	INT;
END_VAR
VAR (* FunctionBlock Status *)
	FBInfoDataDiag	 								AT %I*	:	ARRAY [MIN_FB..MAX_FB] OF UINT; //Safety FB diagnostic information
END_VAR
VAR (* Events/Blocks/Var internal *)
//	EventInputSizeMism										: 	EventHandling := (MsgId:= 1); //Msg id 1 not used for logic terminals
//	EventOutputSizeMism										: 	EventHandling := (MsgId:= 2); //Msg id 1 not used for logic terminals
	EventInvalidCRC											:	EventHandling := (SourceId := DEFAULT_SOURCE_ID, MsgId:= 3);	
	EventCycleCounter										:	EventHandling := (SourceId := DEFAULT_SOURCE_ID, MsgId:= 4);
	EventLogicState											:	EventHandling := (SourceId := DEFAULT_SOURCE_ID, MsgId:= 5);
//	EventDiagHist											:	EventHandling := (SourceId := DEFAULT_SOURCE_ID, MsgId:= 6);
	
//	ReadDiagHist											:	SafetyIODeviceDiagRead;
		
	TON_CycleCounter										:	TON := (PT := TIMEOUT_CYCLE_COUNTER);
	MemCycleCounter											: 	USINT;
	
	EventFBError											:	ARRAY [MIN_FB..MAX_FB] OF EventHandling; //MsgId from 11 to MAX_FB + 10
                        									                        	
	i														:	INT := MIN_FB;

END_VAR

(* EL6910/ ELx9xx Safety Logic Terminal Diag	*)
(************************************************)

(* call IO *************************************************************)
	IO();
	
(* Event 3-10 *******************************************************************)
(* Events 1 and 2 only for EL6900 devices *)

	EventInvalidCRC(
		Flag		:= IO.ProjectCRC = 0 AND_THEN NOT IO.WcState AND IO.InfoDataState = Tc2_EtherCAT.EC_DEVICE_STATE_OP AND Enable,
		ConfirmTrig	:= Quit OR NOT Enable AND EventInvalidCRC.State <> TCEVENTSTATE_INVALID ,
		MsgId		:= ,
		SourceId	:= ,
		Class		:=,
		format		:= ,
		Text1		:= ,
		Text2		:= ,
		pText3		:= ADR(IO.DevName),
		State		=> ,
		Status		=> );
			
	TON_CycleCounter(In  := IO.CycleCounter = MemCycleCounter);
	MemCycleCounter 										:= IO.CycleCounter;   	
	EventCyclecounter(
		Flag		:= TON_CycleCounter.Q AND_THEN NOT IO.WcState AND IO.InfoDataState = Tc2_EtherCAT.EC_DEVICE_STATE_OP AND Enable,
		ConfirmTrig	:= Quit OR NOT Enable AND EventCyclecounter.State <> TCEVENTSTATE_INVALID,
		MsgId		:= ,
		SourceId	:= ,
		Class		:=,
		format		:= ,
		Text1		:= ,
		Text2		:= ,
		pText3		:= ADR(IO.DevName),
		State		=> ,
		Status		=> );	
		
	EventLogicState(
		Flag		:= IO.SafeLogicState = INVALID_SAFETY_LOGIC_STATE AND_THEN NOT IO.WcState AND IO.InfoDataState = Tc2_EtherCAT.EC_DEVICE_STATE_OP AND Enable,
		ConfirmTrig	:= Quit OR NOT Enable AND EventLogicState.State <> TCEVENTSTATE_INVALID ,
		MsgId		:= ,
		SourceId	:= ,
		Class		:=,
		format		:= ,
		Text1		:= ,
		Text2		:= ,
		pText3		:= ADR(IO.DevName),
		State		=> ,
		Status		=> );
		
(* Read error history *********************************************)
(*	ReadDiagHist(
		Busy=> , 
		Done=> , 
		Error=> , 
		ErrorId=> , 
		Execute:= """TBD""" , 
		EcMasterDevId:= , 
		AdsAddr=> , 
		MsgInfoDiag=> , 
		DevType=> , 
		Name=> , 
		FSOEAddr=> , 
		DiagMsgSeverity=> , 
		DiagMsgTextId=> , 
		pDebugData=> , 
		DebugDataMaxId=> );	
		
	EventDiagHist(
		Flag		:= Read.msgSevyIsError AND ReadDiagHist.Done,
		ConfirmTrig	:= Quit OR NOT Enable,
		MsgId		:= ,
		SourceId	:= ,
		Class		:=,
		format		:= ,
		Text1		:= ,
		Text2		:= CONCAT('0x',DWORD_TO_HEXSTR(TO_DWORD(Read.DiagMsgTextId),4,FALSE)),
		pText3		:= ADR(IO.Name),
		State		=> ,
		Status		=> );
*)		
(* Events 11-n FB Error *******************************************)
	NoOfActiveEvents										:= 0;
	Status													:= EventInvalidCRC.Status OR EventCyclecounter.Status OR EventLogicState.status; 

	FOR i := MIN_FB TO MAX_FB 
	DO
		IF FBInfoDataDiag[i] <> 0 AND Enable
			OR EventFBError[i].State <> TCEVENTSTATE_INVALID
		THEN
			EventFBError[i](
				Flag		:= FBInfoDataDiag[i] <> 0 AND Enable,
				ConfirmTrig	:= Quit OR NOT Enable AND EventFBError[i].State <> TCEVENTSTATE_INVALID ,
				MsgId		:= ,
				SourceId	:= ,
				Class		:= ,
				format		:= ,
				Text1		:= ,
				Text2		:= DWORD_TO_BINSTR(TO_DWORD(FBInfoDataDiag[i]),16),
				pText3		:= ADR(IO.DevName),
				State		=> );
			NoOfActiveEvents								:= NoOfActiveEvents + 1;
		END_IF	
		Status												:= Status OR EventFBError[i].Status;
	END_FOR
		

(*********************************************************)

METHOD FB_init : BOOL
VAR_INPUT
	bInitRetains : BOOL; // if TRUE, the retain variables are initialized (warm start / cold start)
	bInCopyCode : BOOL;  // if TRUE, the instance afterwards gets moved into the copy code (online change)
	
END_VAR
	FOR i := MIN_FB TO MAX_FB 
	DO
		EventFBError[i].SourceId 	:= SEL(EventFBError[i].SourceId = 0, EventFBError[i].SourceId, DEFAULT_SOURCE_ID);
		EventFBError[i].MsgId		:= TO_UINT(i + 10);
		EventFBError[i].Text1		:= INT_TO_STRING(i);	
	END_FOR
END_METHOD

PROPERTY PUBLIC sourceId : UDINT
GET
SourceId := EventLogicState.SourceId;
END_GET
SET
IF EventLogicState.SourceId <> SourceId THEN
	EventLogicState.SourceId							:= SourceId;
	EventCycleCounter.SourceId							:= SourceId;
	EventInvalidCRC.SourceId							:= SourceId;
	FOR i := MIN_FB TO MAX_FB 
	DO
		EventFBError[i].SourceId						:= SourceId;
	END_FOR
END_IF
END_SET
END_PROPERTY

END_FUNCTION_BLOCK

// POUs/Safety/Diag/SafetyPlcTerminalDiag
{attribute 'no_check'}
FUNCTION_BLOCK SafetyPlcTerminalDiag // EL6900
VAR CONSTANT
	MIN_FB													:	INT := 1;
	MAX_FB													:	INT := PARAM.SAFETY_PLC_TERM_DIAG_MAX_FB;
END_VAR                 									
VAR_INPUT               									
	Enable													:	BOOL := TRUE;	//FB will be processed as long as enable is TRUE 
	SourceId												:	UDINT := 100300;//Multisource id 
	Quit													:	BOOL;			//Resets error with rising edge 
	IO														:	EL69xx;			
END_VAR
VAR_OUTPUT
	{attribute 'displaymode':='binary'}
	Status													:	DWORD; 			//current sttus of all events
	NoOfActiveEvents										:	INT;
END_VAR
VAR (* FunctionBlock Status *)
	FBInfoDataDiag	 								AT %I*	:	ARRAY [MIN_FB..MAX_FB] OF UINT; //Safety FB diagnostic information
END_VAR
VAR (* Events/Blocks/Var internal *)
	EventInputSizeMism										: EventHandling := (SourceId := SourceId, MsgId:= 1); //Msg id 1
	EventOutputSizeMism										: EventHandling := (SourceId := SourceId, MsgId:= 2); //Msg id 2
	EventInvalidCRC											: EventHandling := (SourceId := SourceId, MsgId:= 3); //Msg id 3
	
	EventFBError											:	ARRAY [MIN_FB..MAX_FB] OF EventHandling; //MsgId from 11 to MAX_FB + 10
                        									                        	
	i														:	INT := MIN_FB;

END_VAR

(* EL6900 Safety Terminal Diag					*)
(************************************************)

(* call IO *************************************************************)
	IO();
	
(* Event 1-10 Size Mismatch ********************************************)
	EventInputSizeMism(
		Flag		:= IO.InputSizeMismatch AND Enable,
		ConfirmTrig	:= Quit OR NOT Enable AND EventInputSizeMism.State <> TCEVENTSTATE_INVALID ,
		MsgId		:= ,
		SourceId	:= ,
		Class		:= ,
		format		:= ,
		Text1		:= ,
		Text2		:= ,
		pText3		:= ,
		State		=> );

	EventOutputSizeMism(
		Flag		:= IO.OutputSizeMismatch AND Enable,
		ConfirmTrig	:= Quit OR NOT Enable AND EventOutputSizeMism.State <> TCEVENTSTATE_INVALID ,
		MsgId		:= ,
		SourceId	:= ,
		Class		:=,
		format		:= ,
		Text1		:= ,
		Text2		:= ,
		pText3		:= ,
		State		=> );
		
	EventInvalidCRC(
		Flag		:= IO.ProjectCRC = 0 AND_THEN NOT IO.WcState AND IO.InfoDataState = Tc2_EtherCAT.EC_DEVICE_STATE_OP AND Enable,
		ConfirmTrig	:= Quit OR NOT Enable AND EventInvalidCRC.State <> TCEVENTSTATE_INVALID ,
		MsgId		:= ,
		SourceId	:= ,
		Class		:=,
		format		:= ,
		Text1		:= ,
		Text2		:= ,
		pText3		:= ,
		State		=> );

	
(* Events 11-n FB Error *******************************************)
	NoOfActiveEvents										:= 0;
	Status													:= EventInputSizeMism.Status OR EventOutputSizeMism.Status OR EventInvalidCRC.Status; 

	FOR i := MIN_FB TO MAX_FB 
	DO
		IF FBInfoDataDiag[i] <> 0 AND Enable
			OR EventFBError[i].State <> TCEVENTSTATE_INVALID
		THEN
			EventFBError[i](
				Flag		:= FBInfoDataDiag[i] <> 0 AND Enable,
				ConfirmTrig	:= Quit OR NOT Enable AND EventFBError[i].State <> TCEVENTSTATE_INVALID ,
				MsgId		:= ,
				SourceId	:= ,
				Class		:= ,
				format		:= ,
				Text1		:= ,
				Text2		:= DWORD_TO_BINSTR(UINT_TO_DWORD(FBInfoDataDiag[i]),16),
				pText3		:= ,
				State		=> );
			NoOfActiveEvents								:= NoOfActiveEvents + 1;
		END_IF	
		Status												:= Status OR EventFBError[i].Status;
	END_FOR

(*********************************************************)

METHOD FB_init : BOOL
VAR_INPUT
	bInitRetains : BOOL; // if TRUE, the retain variables are initialized (warm start / cold start)
	bInCopyCode : BOOL;  // if TRUE, the instance afterwards gets moved into the copy code (online change)
END_VAR

	FOR i := MIN_FB TO MAX_FB 
	DO
		EventFBError[i].MsgId		:= TO_UINT(i + 10);
		EventFBError[i].SourceId	:= SourceId;
		EventFBError[i].Text1		:= INT_TO_STRING(i);	
		EventFBError[i].pText3		:= ADR(IO.DevName);
	END_FOR
END_METHOD

END_FUNCTION_BLOCK

// POUs/Safety/SafetyCircuit
{attribute 'no_check'}
FUNCTION_BLOCK SafetyCircuit (*  *)
VAR_INPUT  
(* periphery Outputs *)
	Demo													:	BOOL := FALSE;		//Return value TRUE = Demo mode for testing
	Enable											AT  %Q*	: 	BOOL := TRUE;		//Enable saftey circuit from PLC - map to first input of AND FB  
	Restart											AT  %Q* :	BOOL;				//Restart safety circuit  - map to restart input of estop/monitoring FB 
                                            	
(* Sequence Times *)                        	
	PT_OnOK													:	TIME := T#3S;
	PT_OnOK_2												:	TIME := T#1S500MS;
	PT_OffOK_2												:	TIME := T#1S500MS;  //be sure that then delay off time is not longer then the safety delay time
END_VAR                                     	
VAR_OUTPUT  
(* periphery Inputs *)      	
	Status													:	SAFETY_CIRCUIT_STATUS;	//Process info from EL69xx                                            	
END_VAR
VAR
	ReadyToRestart									AT  %I*	:	 BOOL; 	//TRUE when restart of safety circuit is executable
	MonOut											AT  %I*	:	 BOOL; 	//Safety estop/monitoring output direct 
	MonDelOut										AT  %I* :	 BOOL;	//Safety estop/monitoring output delay - see EStop/Monitoring FB time settings	
END_VAR
VAR
	TON_OK_1												:	TON;
	TON_OK_2												:	TON;
END_VAR

(* Safetycicrut-control with IOs and stantemachine						*)
(************************************************************************)

(* Safety circuit status *******************************************************)
IF Demo
THEN //Simulation mode 
	CASE status.state OF
	eSTATE.IDLE:	
		TON_OK_1(IN := FALSE); TON_OK_2(IN := FALSE);
		Status.RT											:= FALSE;

	eSTATE.CLEARING:
		TON_OK_2(IN := TRUE, PT := MIN(PT_OnOK_2,PT_OnOK ), Q => Status.OK_2);	
		TON_OK_1(IN := TRUE, PT := PT_OnOK , Q => Status.OK);	
		IF TON_OK_1.Q AND TON_OK_2.Q
		THEN
			Status.RT										:= TRUE;
			status.state 									:= eSTATE.IDLE;
		END_IF
	ELSE
		status.state 										:= eSTATE.CLEARING;
	END_CASE

	Status.FT												:= FALSE;
	Status.InAborting										:= status.state = eSTATE.ABORTING;
	Status.InAborted										:= status.state = eSTATE.ABORTED;
	Status.InClearing										:= status.state = eSTATE.CLEARING;
	Status.InIdle											:= status.state = eSTATE.IDLE;
	
	Status.ReadyToRestart									:= TRUE;
	Status.MonOut											:= TRUE;
	Status.MonDelOut										:= TRUE;
	
ELSE (* statemachine active mode *********************************************************)
	CASE status.state OF
	eSTATE.IDLE:
		status.RT 											:= FALSE;
		IF NOT MonOut OR NOT MonDelOut
		THEN
			TON_OK_1(IN := FALSE); TON_OK_2(IN := FALSE);
			status.state 									:= eSTATE.ABORTING;
		ELSE
			;
		END_IF

	eSTATE.ABORTING:
		IF NOT MonDelOut 
		THEN
			status.OK := status.OK_2 						:= FALSE;
			status.FT 										:= TRUE;
			status.state 									:= eSTATE.ABORTED;
		ELSIF MonOut 
		THEN
			status.FT 										:= TRUE;
			status.state 									:= eSTATE.ABORTED;
		ELSE
			TON_OK_2(IN := TRUE, PT := PT_OffOK_2);
			IF TON_OK_2.Q 
			THEN 
				status.OK_2 								:= FALSE; 
			END_IF
		END_IF

	eSTATE.ABORTED:
		status.FT 											:= FALSE;
		IF 	MonOut AND MonDelOut
		THEN
			TON_OK_1(IN := FALSE); TON_OK_2(IN := FALSE);
			status.state 									:= eSTATE.CLEARING;
		ELSE
			;
		END_IF

	eSTATE.CLEARING:
		IF MonOut AND MonDelOut
		THEN
			TON_OK_1(IN := TRUE, PT := PT_OnOK ,Q => Status.OK );					
			TON_OK_2(IN := TRUE, PT := MIN(PT_OnOK_2,PT_OnOK) ,Q => Status.OK_2);			
			IF status.OK AND status.OK_2 
			THEN
				status.state 								:= eSTATE.IDLE;
				status.RT 									:= TRUE;
			ELSE
				;
			END_IF
		ELSE
			TON_OK_1(IN := FALSE); 
			TON_OK_2(IN := FALSE);
			status.state 									:= eSTATE.ABORTING;
		END_IF
	ELSE
		status.state 										:= eSTATE.ABORTING;
	END_CASE

(* signals *************************************************************)	
	Status.InAborting										:= status.state = eSTATE.ABORTING;
	Status.InAborted										:= status.state = eSTATE.ABORTED;
	Status.InClearing										:= status.state = eSTATE.CLEARING;
	Status.InIdle											:= status.state = eSTATE.IDLE;
                                							
	Status.ReadyToRestart									:= ReadyToRestart;
	Status.MonOut											:= MonOut;
	Status.MonDelOut										:= MonDelOut;		
END_IF

(*********************************************************)

END_FUNCTION_BLOCK

// POUs/Safety/SafetyGroupIO
{attribute 'no_check'}
FUNCTION_BLOCK SafetyGroupIO
VAR_OUTPUT CONSTANT
//Group State
	STATE_UNKNOWN											: BYTE := 0;
	STATE_RUN												: BYTE := 1;
	STATE_STOP												: BYTE := 2;
	STATE_SAFE												: BYTE := 3; //Only EL6900
	STATE_ERROR												: BYTE := 4;
	STATE_RESET												: BYTE := 5;
	STATE_START												: BYTE := 6;
	STATE_STOP_ERROR										: BYTE := 7;
	STATE_DEACTIVE											: BYTE := 16;
	STATE_WAIT_COM_ERROR									: BYTE := 17; 
	
//Group Diag
	DIAG_OK													:	BYTE := 0;
	DIAG_FB_ERROR											:	BYTE := 1;
	DIAG_COM_ERROR											:	BYTE := 2;
	DIAG_MODULE_ERROR										:	BYTE := 3;
	DIAG_CMP_ERROR											:	BYTE := 4;
	DIAG_DEACTIVE_ERROR										:	BYTE := 5;
	DIAG_RESTART_ERROR										:	BYTE := 6;
END_VAR
VAR_INPUT
	ErrAck											AT  %Q*	:	BOOL := FALSE;	//Resets safety group error with rising edge 
	RunStop											AT  %Q* :	BOOL := TRUE;	//TRUE for run and FALSE for stop safety group 
	ModuleFault										AT  %Q* :	BOOL := FALSE;	//

END_VAR                     						
VAR_OUTPUT                  						
	ComErr											AT  %I* : 	BOOL;	//Safety group has a communication error
	ComStartup										AT  %I* :	BOOL;	//Only for EL6910
	FbDeactive										AT  %I* :	BOOL;	//Only for EL6910
	FBErr											AT  %I* : 	BOOL;	//Safety group has a FB error
	FbRun											AT  %I* :	BOOL;	//Only for EL6910
	InRun											AT  %I* :	BOOL;	//Only for EL6910
	OtherErr										AT  %I* :	BOOL;	//Only for EL6910
	OutErr											AT  %I* :	BOOL;	//Safety group has an output error
	
//Only available if the Checkboxes "MapState" and "MapDiag" are selected
	State											AT  %I* : USINT;	//Safety group state - 1=Run/2=Stop/3=Safe/4=Error/5=Reset
	Diag											AT  %I* : USINT;	//Safety group diagnostic information
END_VAR
VAR
END_VAR

(* SafetyGroup IO											             *)
(*************************************************************************)

(*************************************************************************)

{attribute 'monitoring' := 'call'}
PROPERTY Public diagCmpError : bool
GET
DiagCmpError:= Diag = DIAG_CMP_ERROR;
END_GET
END_PROPERTY

{attribute 'monitoring' := 'call'}
PROPERTY Public diagComError : bool
GET
DiagComError:= Diag = DIAG_COM_ERROR;
END_GET
END_PROPERTY

{attribute 'monitoring' := 'call'}
PROPERTY Public diagDeactiveError : bool
GET
DiagDeactiveError:= Diag = DIAG_DEACTIVE_ERROR;
END_GET
END_PROPERTY

{attribute 'monitoring' := 'call'}
PROPERTY PUBLIC diagFbError : BOOL
GET
DiagFbError:= Diag = DIAG_FB_ERROR;;
END_GET
END_PROPERTY

{attribute 'monitoring' := 'call'}
PROPERTY Public diagModuleError : bool
GET
DiagModuleError:= Diag = DIAG_MODULE_ERROR;
END_GET
END_PROPERTY

{attribute 'monitoring' := 'call'}
PROPERTY Public diagNoError : bool
GET
DiagNoError := Diag = 0;
END_GET
END_PROPERTY

{attribute 'monitoring' := 'call'}
PROPERTY Public diagRestartError : bool
GET
DiagRestartError:= Diag = DIAG_RESTART_ERROR;
END_GET
END_PROPERTY

{attribute 'monitoring' := 'call'}
PROPERTY PUBLIC inStateDeactive : bool
GET
inStateDeactive := State = STATE_DEACTIVE;
END_GET
END_PROPERTY

{attribute 'monitoring' := 'call'}
PROPERTY PUBLIC inStateError : BOOL
GET
inStateError :=	State = STATE_ERROR;
END_GET
END_PROPERTY

{attribute 'monitoring' := 'call'}
PROPERTY PUBLIC inStateReset : Bool
GET
inStateReset :=	State = STATE_RESET;
END_GET
END_PROPERTY

{attribute 'monitoring' := 'call'}
PROPERTY PUBLIC inStateRun : BOOL
GET
inStateRun :=	State = STATE_RUN;
END_GET
END_PROPERTY

{attribute 'monitoring' := 'call'}
PROPERTY PUBLIC inStateSafe : Bool
GET
inStateSafe :=	State = STATE_SAFE;
END_GET
END_PROPERTY

{attribute 'monitoring' := 'call'}
PROPERTY PUBLIC inStateStart : Bool
GET
inStateStart :=	State = STATE_START;
END_GET
END_PROPERTY

{attribute 'monitoring' := 'call'}
PROPERTY PUBLIC inStateStop : Bool
GET
inStateStop :=	State = STATE_STOP;
END_GET
END_PROPERTY

{attribute 'monitoring' := 'call'}
PROPERTY PUBLIC inStateStopError : bool
GET
inStateStopError := state = STATE_STOP_ERROR;
END_GET
END_PROPERTY

{attribute 'monitoring' := 'call'}
PROPERTY PUBLIC inStateUnknow : Bool
GET
inStateUnknow :=	State = STATE_UNKNOWN;
END_GET
END_PROPERTY

{attribute 'monitoring' := 'call'}
PROPERTY PUBLIC inStateWaitComError : bool
GET
inStateWaitComError := State = STATE_WAIT_COM_ERROR;
END_GET
END_PROPERTY

END_FUNCTION_BLOCK

// POUs/Safety/SafetyPlcBackupRestore
{attribute 'no_check'}
FUNCTION_BLOCK SafetyPlcBackupRestore Extends FbBase
VAR_OUTPUT CONSTANT
	FNC_BACKUP_EXIST										:	INT := 0; //Check if backup file exists on hardware disk
	FNC_BACKUP												:	INT := 1; //Safe project on hardware disk as hex file
	FNC_RESTORE												:	INT := 2; //Write project back into EL69xx 
END_VAR             										
VAR_INPUT           										
	Fnc														:	INT (FNC_BACKUP_EXIST..FNC_RESTORE) := FNC_BACKUP;
	NetId													: 	T_AmsNetId := '';	//Net ID as text
	EcMasterNetID											: 	T_AmsNetId; 		//AmsNetID of the EtherCAT device *)
	EcMasterPort											: 	T_AmsPort; 			//Port Number of the EL6900 terminal (EtherCAT address) *)
	FilePath												:	T_MaxString := 'C:\'; //path to backup file
	FileName												:	STRING(20) := 'SafetyPlcFW.hex'; //name of backup file                      									
	Timeout													: 	TIME := T#60S;		//time until timeout
END_VAR
VAR_OUTPUT
	DataLength												:	UDINT := 0;
	ErrorFnc												:	STRING(30) := '';
END_VAR
VAR
(* Memory ***********************************************************)
	MemFnc													:	INT := -1;
	
(* Trigger **********************************************************)

(* Timer ************************************************************)
	tonDelay												:	ton;

(* blocks ***********************************************************)
	EnumFindFileEntry										:	FB_EnumFindFileEntry;
	BackupEL6900											:	FB_BackupEL6900;
	RestoreEL6900											:	FB_RestoreEL6900;
	
(* Dummys ***********************************************************)

END_VAR

	(************************************************************************************)
	(*																					*)
	(*		B E C K H O F F   N E W   A U T O M A T I O N   T E C H N O L O G Y    		*)
	(*																					*)
	(*		Eiserstr.5	D-33415 Verl	Germany	phone:	+49-5246-0	www.Beckhoff.Com	*)
    (*																					*)
    (*		Bausteinbeschreibung	:	Restore/Backup plc project 						*)
	(*		TwinCAT-Version			:	3.xx 											*)
	(*		Version					:	V1.1/ 05/16										*)
 	(*		Autor					:	Daniel Schlingmann								*)
	(*		Lib						:	tc2_backuprestoreel6900.compiled-library		*)
	(*																					*)
	(************************************************************************************)

(* Execute ***************************************************************************************)
	rtExecute(CLK := Execute);
	
	CASE state OF
	0:
		Busy												:= FALSE;
		// init		                                	
		IF NOT Execute                              	
		THEN        
			DataLength										:= 0;                                	
			Done 											:= FALSE;
			Error											:= FALSE;
			ErrorID											:= 0;
			ErrorFnc										:= '';
		END_IF                                      			                                            	
		IF rtExecute.Q                             	
		THEN                                        	
			Done 											:= FALSE;
			Busy											:= TRUE;
			Error											:= FALSE;
			ErrorID											:= 0;
			ErrorFnc										:= '';
			DataLength										:= 0;
			MemFnc											:= Fnc;
			BackupEL6900(ReadProject := FALSE);
			RestoreEL6900(writeProject := FALSE);
			EnumFindFileEntry(bExecute := FALSE, sNetId := '', tTimeout := Timeout, sPathName := CONCAT(FilePath,FileName));
			CASE Fnc OF
			FNC_BACKUP_EXIST:state							:= 1;		
			FNC_BACKUP		:state							:= 10;									
			FNC_RESTORE		:state							:= 20;									
			ELSE
				Busy										:= FALSE;
				Done										:= FALSE;
				Error										:= TRUE;
				ErrorId										:= E_AdsErr.DEVICE_INVALIDPARM;	
				ErrorFnc									:= 'SafetyPlcBackupRestore';					
			END_CASE
		END_IF
	
	(* Backup exists *****************************************************)
	1: //first abort old command
		EnumFindFileEntry(bExecute := TRUE ,eCmd := eEnumCmd_Abort );
		IF NOT EnumFindFileEntry.bBusy
		THEN
			EnumFindFileEntry(bExecute := FALSE ,eCmd := eEnumCmd_Abort );
			EnumFindFileEntry(bExecute := TRUE ,eCmd := eEnumCmd_First );
			state											:= State + 1;
		END_IF

	2: //read entrys
		EnumFindFileEntry(bExecute := TRUE);
		IF NOT EnumFindFileEntry.bBusy
		THEN
			IF NOT EnumFindFileEntry.bError
				AND EnumFindFileEntry.stFindFile.sFileName = FileName
			THEN
				Done										:= TRUE;
				Busy										:= FALSE;
				DataLength 									:= EnumFindFileEntry.stFindFile.fileSize.dwLowPart;
				state										:= 0;
			ELSE
				Busy										:= FALSE;
				Done										:= FALSE;
				Error										:= TRUE;
				ErrorId										:= SEL(EnumFindFileEntry.bError , E_AdsErr.DEVICE_NOTFOUND ,EnumFindFileEntry.nErrID);
				ErrorFnc									:= 'EnumFindFileEntry';
				state										:= 0;
			END_IF		
		END_IF
		
	(* Backup (save project to disk) *************************************************************)
	10:
		IF NOT BackupEL6900.bBusy
		THEN
			BackupEL6900(
				ReadProject		:= TRUE, 
				EtherCATAmsNetID:= EcMasterNetID, 
				Port			:= EcMasterPort, 
				FileWriteAmsNetID:= '', 
				FilePathname	:= CONCAT(FilePath,FileName), 
				bBusy			=> , 
				bError			=> , 
				uErrID			=> , 
				ReadDataLength	=> );
			state											:= state + 1;	
		ELSE
			BackupEL6900(ReadProject := FALSE);
		END_IF
		
	11:
		BackupEL6900();
		IF NOT BackupEL6900.bBusy
		THEN
			IF BackupEL6900.bError
			THEN
				Busy										:= FALSE;
				Done										:= FALSE;
				Error										:= TRUE;
				ErrorId										:= BackupEL6900.uErrID;
				ErrorFnc									:= 'BackupEL6900';
				state										:= 0;				
			ELSE
				Done										:= TRUE;
				Busy										:= FALSE;
				DataLength 									:= BackupEL6900.ReadDataLength;	
				state										:= 0;			
			END_IF
		END_IF

	(* Restore *************************************************************)
	20:
		IF NOT RestoreEL6900.bBusy
		THEN
			RestoreEL6900(
				WriteProject	:= TRUE, 
				EtherCATAmsNetID:= EcMasterNetID, 
				Port			:= EcMasterPort, 
				FileReadAmsNetID:= '', 
				FilePathname	:= CONCAT(FilePath,FileName), 
				bBusy			=> , 
				bError			=> , 
				uErrID			=> , 
				WriteDataLength	=> );
			state											:= state + 1;	
		ELSE
			RestoreEL6900(WriteProject := FALSE);
		END_IF
		
	21:
		RestoreEL6900();
		IF NOT RestoreEL6900.bBusy
		THEN
			IF RestoreEL6900.bError
			THEN
				Busy										:= FALSE;
				Done										:= FALSE;
				Error										:= TRUE;
				ErrorId										:= RestoreEL6900.uErrID;
				ErrorFnc									:= 'RestoreEL6900';
				state										:= 0;				
			ELSE
				Done										:= TRUE;
				Busy										:= FALSE;
				DataLength 									:= RestoreEL6900.WriteDataLength;	
				state										:= 0;			
			END_IF
		END_IF
		
	END_CASE
			
(*************************************************************************************************)

METHOD PUBLIC backup : BOOL //Return value = TRUE if busy
//required parameter
//EcMasterNetID
//EcMasterPort
//FilePath
VAR_INPUT
	Execute													:	BOOL;
END_VAR
CASE state OF
0:	
	Fnc 													:= FNC_BACKUP;
	THIS^(Execute:=Execute);
1: 
	;

END_CASE
Backup 														:= Busy;
END_METHOD

METHOD PUBLIC fileExists : BOOL //Return value = TRUE if busy
//required parameter
//FilePath
VAR_INPUT
	Execute													:	BOOL;
END_VAR
CASE state OF
0:	
	Fnc 													:= FNC_BACKUP_EXIST;
	THIS^(Execute:=Execute);
1: 
	;

END_CASE
fileExists 														:= Busy;
END_METHOD

METHOD PUBLIC restore : BOOL //Return value = TRUE if busy
//required parameter
//EcMasterNetID
//EcMasterPort
//FilePath
VAR_INPUT
	Execute													:	BOOL;
END_VAR
CASE state OF
0:	
	Fnc 													:= FNC_RESTORE;
	THIS^(Execute:=Execute);
1: 
	;

END_CASE
Restore 													:= Busy;
END_METHOD

END_FUNCTION_BLOCK

// POUs/StringHelper/ExtendedString/ExtString
{attribute 'no_check' := ''}
FUNCTION_BLOCK ExtString //STRING functions for a string with a lenght > 255. Lenght is defined by PARAM.MAX_EXT_STRING_LENGTH
VAR_OUTPUT CONSTANT
	MAX_LENGTH												: UDINT := PARAM.MAX_EXT_STRING_LENGTH;
END_VAR
VAR_OUTPUT
	ResultStr												: T_EXT_STRING;		
END_VAR
VAR									
	str1Len													: UDINT;
 	str2Len													: UDINT; 
	cpyLenght												: UDINT;
END_VAR

//Concatenation (combination) of two extended strings (lenght definded by ET.Param.EXT_STRING_MAX_LENGHT)
METHOD CONCAT : UDINT //Returns the lenght of the new string
VAR_INPUT
	 rSTR1													:	REFERENCE TO T_EXT_STRING;
	 STR2													:	T_EXT_STRING;
	 rResult												:	REFERENCE TO T_EXT_STRING;
END_VAR
VAR_OUTPUT
END_VAR
VAR
END_VAR
MEMSET(ADR(ResultStr),0,SIZEOF(ResultStr));
IF __ISVALIDREF(rSTR1) 
THEN
	str1Len 													:= LEN(rSTR1);
	str2Len 													:= LEN(STR2);
	MEMCPY(ADR(ResultStr), ADR(rSTR1), str1Len + 1);	 //Copy first string to result
	cpyLenght													:= 1 + MIN(str2Len, MAX_LENGTH - str1Len);
	MEMCPY(ADR(ResultStr) + str1Len, ADR(STR2), SEL(cpyLenght >  1, 0, cpyLenght)); //Add second string
	CONCAT														:= MIN(str1Len + str2Len,MAX_LENGTH);
	IF __ISVALIDREF(rResult) 
	THEN
		MEMCPY(ADR(rResult), ADR(ResultStr), CONCAT + 1); 
	END_IF
ELSE
	CONCAT														:= 0;
END_IF
END_METHOD

//The function DELETE removes a partial STRING from a larger STRING at a defined position. 
//The input variable rSTR is TYPE STRING with a lenght if ET.Param.EXT_STRING_MAX_LENGHT, LEN AND POS are TYPE UINT.
//The new string will be written into the result reference, in case of invalid pos or len parameter, the input string will be copied to rResult
//means: Delete LEN characters from rSTR beginning with the character in the POS
METHOD PUBLIC DELETE : UDINT //Returns the new string lenght
VAR_INPUT
	 rSTR													:	REFERENCE TO T_EXT_STRING;
	 LEN													:	UDINT (0..MAX_LENGTH) := 0;
	 POS													:	UDINT (0..MAX_LENGTH) := 0;
	 rResult												:	REFERENCE TO T_EXT_STRING;						
END_VAR
VAR
END_VAR
MEMSET(ADR(ResultStr),0,SIZEOF(ResultStr));
IF NOT __ISVALIDREF(rSTR)  
THEN
	DELETE													:= 0;
	RETURN;
END_IF
Str1Len 													:= THIS^.LEN(rSTR);
IF pos > 0 AND pos <= str1Len
THEN // Only executed if parameter within string limitation
	MEMCPY(ADR(ResultStr), ADR(rStr), MAX(0, POS -1 )); //First part of string
	cpyLenght 												:= Str1Len - MIN(Str1Len, MAX(0, POS -1 ) + LEN); 
	MEMCPY(ADR(ResultStr) + MAX(0,POS-1), ADR(rStr) + MIN(Str1Len, POS -1 + LEN), cpyLenght + 1); //Second part of string
	DELETE													:= (cpyLenght - 1) + pos; //New string length
	IF __ISVALIDREF(rResult) 
	THEN
		MEMCPY(ADR(rResult), ADR(ResultStr), DELETE + 1); 
	END_IF
ELSE
	DELETE													:= Str1Len;
	IF __ISVALIDREF(rResult) 
	THEN
		MEMMOVE(ADR(rResult), ADR(rSTR), DELETE + 1); 
	END_IF	
END_IF
END_METHOD

//FIND searches for a partial string within a string. FIND(STR1, STR2) 
//means: Find the position of the first character where STR2 appears in STR1 for the first time. 
//If STR2 is not found in STR1, then FIND:=0.
METHOD PUBLIC FIND : UDINT //position of the first character where STR2 appears in STR1 for the first time.
VAR_INPUT
	 rSTR1													: REFERENCE TO T_EXT_STRING;
	 STR2													: T_EXT_STRING;
END_VAR
VAR
	 valid													: BOOL;
	 i, j													: UDINT;
END_VAR
FIND														:= 0;
IF NOT __ISVALIDREF(rSTR1)
THEN
	RETURN;
END_IF

str1Len 													:= LEN(rSTR1);
str2Len 													:= LEN(STR2);
FOR i:= 0 TO str1Len 
DO
	IF rSTR1[i] = STR2[0] 
	THEN	// Wenn erstes Zeichen übereinstimmt
		valid												:= TRUE;
		FOR j := 1 TO str2Len - 1 DO // Alle zeichen von STR2 durchgehen
			valid 											:= rSTR1[i + j] = STR2[j];
			
			IF NOT valid THEN // Wenn Zeichen ungleich abbrechen
				RETURN;						
			END_IF	
		END_FOR
		FIND 											:= i + 1;
		RETURN;		
	END_IF
END_FOR
END_METHOD

//INSERT inserts a string into another string at a defined point.
//means: insert STR2 into STR1 after position POS.
METHOD PUBLIC INSERT : UDINT //Returns the lenght of the new string
VAR_INPUT
	 rSTR1													: REFERENCE TO T_EXT_STRING;
	 STR2													: T_EXT_STRING;
	 POS													: UDINT (0..MAX_LENGTH);  
	 rResult												: REFERENCE TO T_EXT_STRING;	
END_VAR
VAR
	 chkPos													: UDINT;	
END_VAR
MEMSET(ADR(ResultStr),0,SIZEOF(ResultStr));
IF NOT __ISVALIDREF(rSTR1) 
THEN
	INSERT														:= 0;
	RETURN;
END_IF
str1Len 													:= LEN(rSTR1);
str2Len 													:= LEN(STR2);
IF Pos >= 0 AND Pos <= Str1Len
THEN
	MEMCPY(ADR(ResultStr), ADR(rStr1), str1Len + 1);  //Copy string to to result
	chkPos 													:= LIMIT(0, POS, str1Len); //Limit insert pos to lenght string 1
	cpyLenght												:= MAX(0,MIN(str1Len - chkPos  + 1, MAX_LENGTH - chkPos - str2Len));
	MEMCPY(ADR(ResultStr) + chkPos + str2Len, ADR(rResult) + chkPos,SEL(cpyLenght > 1, 0,cpyLenght)); //move rest of string 1 to the end
	cpyLenght												:= MIN(str2Len , MAX_LENGTH - chkPos);
	MEMCPY(ADR(ResultStr) + chkPos, ADR(Str2) ,cpyLenght );
	INSERT													:= MIN(MAX_LENGTH, str1Len + str2Len);
	IF __ISVALIDREF(rResult) 
	THEN
		MEMCPY(ADR(rResult), ADR(ResultStr), INSERT + 1); 
	END_IF
ELSE
	INSERT													:= str1Len;
	IF __ISVALIDREF(rResult) 
	THEN
		MEMMOVE(ADR(rResult), ADR(rStr1), INSERT + 1); 
	END_IF
END_IF
END_METHOD

//Left returns the left, initial string for a given string. LEFT (STR, SIZE) 
//means: Take the first SIZE character from the right in the string STR.
METHOD PUBLIC LEFT : UDINT
VAR_INPUT
	 rSTR													: REFERENCE TO T_EXT_STRING;
	 SIZE													: UDINT (0..MAX_LENGTH);
	 rResult												: REFERENCE TO T_EXT_STRING;
END_VAR
VAR_INPUT
	 
END_VAR
MEMSET(ADR(ResultStr),0,SIZEOF(ResultStr));
IF __ISVALIDREF(rSTR)
THEN
	SIZE													:= LIMIT(0,SIZE,MAX_LENGTH); 
	LEFT													:= MIN(LEN(rSTR), SIZE);
	MEMCPY(ADR(ResultStr), ADR(rSTR), LEFT);	
	IF __ISVALIDREF(rResult) 
	THEN
		MEMCPY(ADR(rResult), ADR(ResultStr), LEFT + 1); 
	END_IF
ELSE
	LEFT													:= 0;
END_IF
END_METHOD

//Returns the length of a string.
METHOD PUBLIC LEN : UDINT
VAR_INPUT
	rSTR												:	REFERENCE TO T_EXT_STRING;
END_VAR
VAR
	i													:	UDINT;
END_VAR
IF __ISVALIDREF(rSTR) 
THEN
	LEN														:= 0;								
	FOR i := 0 TO MAX_LENGTH 
	DO
		IF rSTR[i] = 0 
		THEN
			LEN 											:= i;
			RETURN;
		END_IF
	END_FOR
ELSE
	LEN														:= 0;
END_IF
END_METHOD

//Mid returns a partial string from within a string. MID (STR, LEN, POS) 
//means: Retrieve LEN characters from the STR string beginning with the character at position POS.
METHOD PUBLIC MID : UDINT //Returns the lenght if the new string (result)
VAR_INPUT
	 rSTR													:	REFERENCE TO T_EXT_STRING;
	 LEN													:	UDINT (0..MAX_LENGTH) ;
	 POS													:	UDINT (0..MAX_LENGTH) ;
	 rResult												:	REFERENCE TO T_EXT_STRING;	
END_VAR
VAR
END_VAR
MEMSET(ADR(ResultStr),0,SIZEOF(ResultStr));
IF NOT __ISVALIDREF(rSTR)
THEN
	MID														:= 0;
	RETURN;	
END_IF

str1Len 													:= THIS^.LEN(rSTR);

IF POS >= 0 AND POS <= str1Len 
THEN	 
	cpyLenght 												:= MIN(str1Len - POS + 1, MIN(LEN, str1Len));	
	MEMCPY(ADR(ResultStr), ADR(rSTR) + MAX(0,POS -1), cpyLenght);
	MID														:= cpyLenght;
	IF __ISVALIDREF(rResult) 
	THEN
		MEMCPY(ADR(rResult), ADR(ResultStr), MID + 1); 
	END_IF
ELSE
	MID														:= str1Len;
	IF __ISVALIDREF(rResult) 
	THEN
		MEMMOVE(ADR(rResult), ADR(rStr), MID + 1); 
	END_IF	
END_IF
END_METHOD

//REPLACE replaces a partial string from a larger string with a third string. REPLACE(STR1, STR2, L, P) 
//means: Replace LEN characters from STR1 with STR2 beginning with the character in the position POS.
METHOD PUBLIC REPLACE : UDINT
VAR_INPUT
	 rSTR1													:	REFERENCE TO T_EXT_STRING;
	 STR2													:	T_EXT_STRING;
	 LEN													:	UDINT (0..MAX_LENGTH);
	 POS													:	UDINT (0..MAX_LENGTH);
	 rResult												:	REFERENCE TO T_EXT_STRING;
END_VAR
VAR
END_VAR
MEMSET(ADR(ResultStr),0,SIZEOF(ResultStr));
IF __ISVALIDREF(rSTR1) 
THEN	
	str1Len 												:= THIS^.LEN(rSTR1);
	str2Len 												:= THIS^.LEN(STR2);
	
	Pos														:= LIMIT(0,Pos -1, Str1Len);
	Len														:= LIMIT(0,Len,str1Len);
	MEMCPY(ADR(ResultStr), ADR(rSTR1), Pos); //Copy first part of string 
	MEMCPY(ADR(ResultStr) + Pos , ADR(STR2), MIN(str2Len + 1, MAX_LENGTH - Pos )); //insert string two
 	cpyLenght 												:= MAX(0,MIN(str1Len - Pos - Len, MAX_LENGTH - str2Len - Pos));
	MEMCPY(ADR(ResultStr) + Pos + str2Len, ADR(rSTR1) + Pos + Len, SEL(cpyLenght > 1, 0,cpyLenght));	//Add rest if string 1
	REPLACE 												:= MIN(MAX_LENGTH, Str2Len + pos + MAX(0,Str1Len - Len - Pos));
	IF __ISVALIDREF(rResult) 
	THEN
		MEMCPY(ADR(rResult), ADR(ResultStr), REPLACE + 1); 
	END_IF	
ELSE
	REPLACE 												:= 0;
END_IF
END_METHOD

//Right returns the right, initial string for a given string. RIGHT (STR, SIZE) 
//means: Take the first SIZE character from the right in the string STR.
METHOD PUBLIC RIGHT : UDINT
VAR_INPUT
	 rSTR													: REFERENCE TO T_EXT_STRING;
	 SIZE													: UDINT (0..MAX_LENGTH);
	 rResult												: REFERENCE TO T_EXT_STRING;
END_VAR
VAR
	 chkSize												: UDINT;
END_VAR
MEMSET(ADR(ResultStr),0,SIZEOF(ResultStr));
IF __ISVALIDREF(rSTR)
THEN
	str1Len 												:= LEN(rSTR);
	chkSize 												:= MIN(str1Len,MIN(MAX_LENGTH, SIZE));
	MEMCPY(ADR(ResultStr), ADR(rSTR) + str1Len - chkSize, chkSize + 1);
	RIGHT													:= chkSize;
	IF __ISVALIDREF(rResult) 
	THEN
		MEMCPY(ADR(rResult), ADR(ResultStr), RIGHT + 1); 
	END_IF	
ELSE
	RIGHT													:= 0;
END_IF
END_METHOD

END_FUNCTION_BLOCK

// POUs/StringHelper/ExtendedString/ExtWString
{attribute 'no_check' := ''}
FUNCTION_BLOCK ExtWString //WSTRING functions for a wstring with a lenght > 255. Lenght is defined by PARAM.MAX_EXT_STRING_LENGTH
VAR_OUTPUT CONSTANT
	MAX_LENGTH												: UDINT := PARAM.MAX_EXT_STRING_LENGTH;
END_VAR
VAR_OUTPUT
	ResultStr												: T_EXT_WSTRING;		
END_VAR
VAR
	str1Len													: UDINT;
 	str2Len													: UDINT; 
	cpyLenght												: UDINT;
END_VAR

//Concatenation (combination) of two extended wstrings (lenght definded by ET.Param.EXT_STRING_MAX_LENGHT)
METHOD CONCAT : UDINT //Returns the lenght of the new string
VAR_INPUT
	 rSTR1													:	REFERENCE TO T_EXT_WSTRING;
	 STR2													:	T_EXT_WSTRING;
	 rResult												:	REFERENCE TO T_EXT_WSTRING;
END_VAR
VAR_OUTPUT
END_VAR
VAR
END_VAR
MEMSET(ADR(ResultStr),0,SIZEOF(ResultStr));
IF __ISVALIDREF(rSTR1)
THEN
	str1Len 													:= LEN(rSTR1);
	str2Len 													:= LEN(STR2);
	MEMCPY(ADR(ResultStr), ADR(rSTR1), (str1Len + 1) * 2);	 //Copy first string to result
	cpyLenght													:= 1 + MIN(str2Len, MAX_LENGTH - str1Len);
	MEMCPY(ADR(ResultStr) + (2 * str1Len), ADR(STR2), SEL(cpyLenght >  1, 0, cpyLenght) * 2); //Add second string
	CONCAT														:= MIN(str1Len + str2Len,MAX_LENGTH);
	IF __ISVALIDREF(rResult) 
	THEN
		MEMCPY(ADR(rResult), ADR(ResultStr), 2 * (CONCAT + 1)); 
	END_IF
ELSE
	CONCAT														:= 0;
END_IF
END_METHOD

//The function DELETE removes a partial STRING from a larger WSTRING at a defined position. 
//The input variable rSTR is TYPE WSTRING with a lenght if ET.Param.EXT_STRING_MAX_LENGHT, LEN AND POS are TYPE UINT.
//The new string will be written into the result reference, in case of invalid pos or len parameter, the input string will be copied to rResult
//means: Delete LEN characters from rSTR beginning with the character in the POS
METHOD PUBLIC DELETE : UDINT //Returns the new string lenght
VAR_INPUT
	 rSTR													:	REFERENCE TO T_EXT_WSTRING;
	 LEN													:	UDINT (0..MAX_LENGTH) := 0;
	 POS													:	UDINT (0..MAX_LENGTH) := 0;
	 rResult												:	REFERENCE TO T_EXT_WSTRING;						
END_VAR
VAR
END_VAR
MEMSET(ADR(ResultStr),0,SIZEOF(ResultStr));
IF NOT __ISVALIDREF(rSTR) 
THEN
	DELETE													:= 0;
	RETURN;
END_IF

Str1Len 													:= THIS^.LEN(rSTR);
IF pos > 0 AND pos <= str1Len
THEN // Only executed if parameter within string limitation
	MEMCPY(ADR(ResultStr), ADR(rStr), MAX(0, POS -1 ) * 2); //First part of string
	cpyLenght 												:= Str1Len - MIN(Str1Len, MAX(0, POS -1 ) + LEN); 
	MEMCPY(ADR(ResultStr) + (2 * MAX(0,POS-1)), ADR(rStr) + (2 * MIN(Str1Len, POS -1 + LEN)), (cpyLenght + 1) * 2); //Second part of string
	DELETE													:= (cpyLenght - 1) + pos; //New string length
	IF __ISVALIDREF(rResult) 
	THEN
		MEMCPY(ADR(rResult), ADR(ResultStr), 2 * (DELETE + 1)); 
	END_IF
ELSE
	DELETE													:= Str1Len;
	IF __ISVALIDREF(rResult) 
	THEN
		MEMMOVE(ADR(rResult), ADR(rStr), 2 * (DELETE + 1)); 
	END_IF	
END_IF
END_METHOD

//FIND searches for a partial wstring within a wstring. FIND(STR1, STR2)
//means: Find the position of the first character where STR2 appears in STR1 for the first time. 
//If STR2 is not found in STR1, then FIND:=0.
METHOD PUBLIC FIND : UDINT //position of the first character where STR2 appears in STR1 for the first time.
VAR_INPUT
	 rSTR1													: REFERENCE TO T_EXT_WSTRING;
	 STR2													: T_EXT_WSTRING;
END_VAR
VAR
	 valid													: BOOL;
	 i, j													: UDINT;
END_VAR
FIND														:= 0;
IF NOT __ISVALIDREF(rSTR1) 
THEN
	RETURN;
END_IF

str1Len 													:= LEN(rSTR1);
str2Len 													:= LEN(STR2);
FOR i:= 0 TO str1Len 
DO
	IF rSTR1[i] = STR2[0] 
	THEN	// Wenn erstes Zeichen übereinstimmt
		valid												:= TRUE;
		FOR j := 1 TO str2Len - 1 DO // Alle zeichen von STR2 durchgehen
			valid 											:= rSTR1[i + j] = STR2[j];
			
			IF NOT valid THEN // Wenn Zeichen ungleich abbrechen
				RETURN;						
			END_IF	
		END_FOR
		FIND 												:= i + 1;
		RETURN;		
	END_IF
END_FOR
END_METHOD

//INSERT inserts a string into another wstring at a defined point.
//means: insert STR2 into STR1 after position POS.
METHOD PUBLIC INSERT : UDINT //Returns the lenght of the new string
VAR_INPUT
	 rSTR1													: REFERENCE TO T_EXT_WSTRING;
	 STR2													: T_EXT_WSTRING;
	 POS													: UDINT (0..MAX_LENGTH);  
	 rResult												: REFERENCE TO T_EXT_WSTRING;	
END_VAR
VAR
	 chkPos													: UDINT;	
END_VAR
MEMSET(ADR(ResultStr),0,SIZEOF(ResultStr));
IF NOT __ISVALIDREF(rSTR1) 
THEN
	INSERT													:= 0;
	RETURN;
END_IF
str1Len 													:= LEN(rSTR1);
str2Len 													:= LEN(STR2);
IF Pos >= 0 AND Pos <= Str1Len
THEN
	MEMCPY(ADR(ResultStr), ADR(rStr1), 2* (str1Len + 1));  //Copy string to to result
	chkPos 													:= LIMIT(0, POS, str1Len); //Limit insert pos to lenght string 1
	cpyLenght												:= MAX(0,MIN(str1Len - chkPos  + 1, MAX_LENGTH - chkPos - str2Len));
	MEMCPY(ADR(ResultStr) + (2 * (chkPos + str2Len)), ADR(rResult) + (2 * chkPos) ,2 * SEL(cpyLenght > 1, 0,cpyLenght)); //move rest of string 1 to the end
	cpyLenght												:= MIN(str2Len , MAX_LENGTH - chkPos);
	MEMCPY(ADR(ResultStr) + (2 * chkPos), ADR(Str2) ,cpyLenght * 2 );
	INSERT													:= MIN(MAX_LENGTH, str1Len + str2Len);
	IF __ISVALIDREF(rResult) 
	THEN
		MEMCPY(ADR(rResult), ADR(ResultStr), 2 * (INSERT + 1)); 
	END_IF
ELSE
	INSERT													:= str1Len;
	IF __ISVALIDREF(rResult) 
	THEN
		MEMMOVE(ADR(rResult), ADR(rStr1), 2 * (INSERT + 1)); 
	END_IF; 
END_IF
END_METHOD

//Left returns the left, initial wstring for a given string. LEFT (STR, SIZE) 
//means: Take the first SIZE character from the left in the string STR.
METHOD PUBLIC LEFT : UDINT
VAR_INPUT
	 rSTR													: REFERENCE TO T_EXT_WSTRING;
	 SIZE													: UDINT (0..MAX_LENGTH);
	 rResult												: REFERENCE TO T_EXT_WSTRING;
END_VAR
VAR_INPUT
	 
END_VAR
MEMSET(ADR(ResultStr),0,SIZEOF(ResultStr));
IF __ISVALIDREF(rSTR)
THEN
	SIZE													:= LIMIT(0,SIZE,MAX_LENGTH); 
	LEFT													:= MIN(LEN(rSTR), SIZE);
	MEMCPY(ADR(ResultStr), ADR(rSTR), 2 * LEFT);
	IF __ISVALIDREF(rResult) 
	THEN
		MEMCPY(ADR(rResult), ADR(ResultStr), 2 * (LEFT + 1)); 
	END_IF
ELSE
	LEFT													:= 0;
END_IF
END_METHOD

//Returns the length of a extended wstring.
METHOD PUBLIC LEN : UDINT
VAR_INPUT
	rSTR												:	REFERENCE TO T_EXT_WSTRING;
END_VAR
VAR
	i													:	UDINT;
END_VAR
IF __ISVALIDREF(rSTR) 
THEN
	LEN														:= 0;								
	FOR i := 0 TO MAX_LENGTH 
	DO
		IF rSTR[i] = 0 
		THEN
			LEN 											:= i;
			RETURN;
		END_IF
	END_FOR
ELSE
	LEN														:= 0;
END_IF
END_METHOD

//Mid returns a partial string from within a wstring. MID (STR, LEN, POS) 
//means: Retrieve LEN characters from the STR string beginning with the character at position POS.
METHOD PUBLIC MID : UDINT //Returns the lenght if the new string (result)
VAR_INPUT
	 rSTR													:	REFERENCE TO T_EXT_WSTRING;
	 LEN													:	UDINT (0..MAX_LENGTH) ;
	 POS													:	UDINT (0..MAX_LENGTH) ;
	 rResult												:	REFERENCE TO T_EXT_WSTRING;	
END_VAR
VAR
END_VAR
MEMSET(ADR(ResultStr),0,SIZEOF(ResultStr));
IF NOT __ISVALIDREF(rSTR)
THEN
	MID														:= 0;
	RETURN;	
END_IF

str1Len 													:= THIS^.LEN(rSTR);

IF POS >= 0 AND POS <= str1Len 
THEN	 
	cpyLenght 												:= MIN(str1Len - POS + 1, MIN(LEN, str1Len));	
	MEMMOVE(ADR(ResultStr), ADR(rSTR) + (2 * MAX(0,POS -1)), 2 * cpyLenght);
	MID														:=  cpyLenght;
	IF __ISVALIDREF(rResult) 
	THEN
		MEMCPY(ADR(rResult), ADR(ResultStr), 2 * (MID + 1)); 
	END_IF
ELSE
	IF __ISVALIDREF(rResult) 
	THEN
		MEMMOVE(ADR(rResult), ADR(rStr), 2 * (str1Len + 1)); 
	END_IF
	MID														:= str1Len;
END_IF
END_METHOD

//REPLACE replaces a partial wstring from a larger wstring with a third wstring. REPLACE(STR1, STR2, L, P) 
//means: Replace LEN characters from STR1 with STR2 beginning with the character in the position POS.
METHOD PUBLIC REPLACE : UDINT
VAR_INPUT
	 rSTR1													:	REFERENCE TO T_EXT_WSTRING;
	 STR2													:	T_EXT_WSTRING;
	 LEN													:	UDINT (0..MAX_LENGTH);
	 POS													:	UDINT (0..MAX_LENGTH);
	 rResult												:	REFERENCE TO T_EXT_WSTRING;
END_VAR
VAR
END_VAR
MEMSET(ADR(ResultStr),0,SIZEOF(ResultStr));
IF __ISVALIDREF(rSTR1) 
THEN	
	str1Len 												:= THIS^.LEN(rSTR1);
	str2Len 												:= THIS^.LEN(STR2);
	
	Pos														:= LIMIT(0,Pos -1, Str1Len);
	Len														:= LIMIT(0,Len,str1Len);
	MEMCPY(ADR(ResultStr), ADR(rSTR1), 2 * Pos); //Copy first part of string 
	MEMCPY(ADR(ResultStr) + (2 * Pos) , ADR(STR2), 2 * (MIN(str2Len + 1, MAX_LENGTH - Pos ))); //insert string two
 	cpyLenght 												:= MAX(0,MIN(str1Len - Pos - Len, MAX_LENGTH - str2Len - Pos));
	MEMCPY(ADR(ResultStr) + (2 * (Pos + str2Len)), ADR(rSTR1) + (2 * (Pos + Len)), 2 * SEL(cpyLenght > 1, 0,cpyLenght));	//Add rest if string 1
	REPLACE 												:= MIN(MAX_LENGTH, Str2Len + pos + MAX(0,Str1Len - Len - Pos));
	IF __ISVALIDREF(rResult) 
	THEN
		MEMMOVE(ADR(rResult), ADR(ResultStr), 2 * (REPLACE + 1)); 
	END_IF	
ELSE
	REPLACE 												:= 0;
END_IF
END_METHOD

//Right returns the right, initial string for a given wstring. RIGHT (STR, SIZE) 
//means: Take the first SIZE character from the right in the string STR.
METHOD PUBLIC RIGHT : UDINT
VAR_INPUT
	 rSTR													: REFERENCE TO WSTRING(MAX_LENGTH);
	 SIZE													: UDINT (0..MAX_LENGTH);
	 rResult												: REFERENCE TO WSTRING(MAX_LENGTH);
END_VAR
VAR
	 chkSize												: UDINT;
END_VAR
MEMSET(ADR(ResultStr),0,SIZEOF(ResultStr));
IF __ISVALIDREF(rSTR)
THEN
	str1Len 												:= LEN(rSTR);
	chkSize 												:= MIN(str1Len,MIN(MAX_LENGTH, SIZE));
	MEMCPY(ADR(ResultStr), ADR(rSTR) + (2 * (str1Len - chkSize)), 2* ( chkSize + 1));
	RIGHT													:= chkSize;
	IF __ISVALIDREF(rResult) 
	THEN
		MEMCPY(ADR(rResult), ADR(ResultStr), 2 * (RIGHT + 1)); 
	END_IF	
ELSE
	RIGHT													:= 0;
END_IF
END_METHOD

END_FUNCTION_BLOCK

// POUs/StringHelper/cutStrNumberToSeperator
{attribute 'no_check'}
//Cut "number" from left site of string. Value will be written into LREAL Target variable in case found string is a valid number
//Function return value will be S_OK if a number is found, S_FALSE if string is empty and E_HRESULTADSERR.ERROR in case found characters are not a number
//Attention! do not use variables smaller then T_MaxString for Source parameter
FUNCTION cutStrNumberToSeperator : HRESULT
VAR_INPUT
	Seperator									:	STRING(5);
END_VAR
VAR_IN_OUT
	Source										:	T_MAXSTRING;
	Target										:	LREAL;
END_VAR
VAR
	tmpString									:	STRING;
	pSource										:	POINTER TO 	T_MAXSTRING;
END_VAR


	pSource										:= ADR(Source);
	tmpString									:= cutStrToSeperator(Seperator, pSource^);
	IF tmpString[0] = 0
	THEN
		cutStrNumberToSeperator					:= S_FALSE;				
	ELSIF isStringNumeric(ADR(tmpString)) 
	THEN 
		Target 									:= TO_LREAL(tmpString); 
	
		cutStrNumberToSeperator					:= S_OK;
	ELSE 
		cutStrNumberToSeperator					:= E_HRESULTADSERR.ERROR;
	END_IF

END_FUNCTION

// POUs/StringHelper/cutStrToSeperator
{attribute 'no_check'}
//Returns string found on left site of seperator and cut of the return part from the origin string, empty if seperator is not found
//Attention! do not use variables smaller then T_MaxString for strline parameter or return value of function
FUNCTION cutStrToSeperator : T_MaxString
VAR_INPUT
	Seperator												:	STRING(10) :=';';
END_VAR             										
VAR_IN_OUT         										
	Strline													:	T_MaxString;
END_VAR             										
VAR       
	lenght,pos												:	INT;          	
	tmp														:	T_MaxString;
END_VAR

IF strline = '' 
THEN
	cutStrToSeperator										:= strline;
ELSE
	pos 													:= FIND (strline,seperator);
	IF pos > 0 
	THEN
		cutStrToSeperator									:= LEFT(strline,pos-1);	
		Lenght												:= LEN(strline);	
		IF Lenght > pos 
		THEN //write back string without seperator		
			tmp												:= RIGHT(strline, Lenght - (pos - 1 + LEN(seperator))); //Save rest
			MEMSET(ADR(strline), 0, TO_UDINT(Lenght));//delete complete string
			MEMCPY(ADR(strline), ADR(tmp), TO_UDINT(LEN(tmp)));
		ELSE //Delete stringline because seperator is at the end
			MEMSET(ADR(strline), 0, TO_UDINT(Lenght));//delete complete string
		END_IF              								
	ELSE                    								
		cutStrToSeperator									:='';
	END_IF
END_IF

END_FUNCTION

// POUs/StringHelper/isStringNumeric
{attribute 'no_check'}
//Returns TRUE in case a ascii string contains only a valid number signs. Minus,plus,space,comma and dot are allowed
//Limited to a Param.MAX_EXT_STRING_LENGTH long string  
FUNCTION isStringNumeric : BOOL 
VAR_INPUT
	pSource													:	POINTER TO BYTE;
END_VAR             										
VAR                 
	Char													:	BYTE;										
	countSeperator											:	INT;
	i														:	UDINT;
	Addr													:	POINTER TO BYTE;
END_VAR

IF pSource <> 0
THEN
	isStringNumeric											:=	TRUE;
	FOR i := 0 TO PARAM.MAX_EXT_STRING_LENGTH DO
		Addr												:= pSource + i;
		Char												:= Addr^;
		IF Char = 0
		THEN
			isStringNumeric									:= i > 0; //Only TRUE if string is not empty 
			EXIT;
		ELSIF Char = 46 OR Char = 44 //comma or point as a seperator
		THEN
			countSeperator									:= countSeperator + 1;
			IF countSeperator > 1 
			THEN
				isStringNumeric								:= FALSE;
				EXIT;	(* more than one seperator -> no number *)
			END_IF
		ELSIF(Char < 48 OR Char > 57)
			AND Char <> 45 (* minus *)
			AND Char <> 43 (* plus *)
			AND Char <> 32 (* Space *)
			AND Char <> 101(* e for 9.9999992e-2 *)
			OR i = PARAM.MAX_EXT_STRING_LENGTH
		THEN
			isStringNumeric									:= FALSE;
			EXIT;	(* no numerical char *)
		END_IF
	END_FOR      
ELSE
	isStringNumeric											:= FALSE;
END_IF

END_FUNCTION

// POUs/StringHelper/cutWStrToSeperator
{attribute 'no_check'}
//Returns string found on left site of seperator and cut of the return part from the origin string, empty if seperator is not found
//Attention! do not use variables smaller then T_MaxString for strline parameter or return value of function
FUNCTION cutWStrToSeperator : WSTRING(MAX_STRING_LENGTH)
VAR_INPUT
	Seperator												:	WSTRING(10) :=";";
END_VAR             										
VAR_IN_OUT         										
	Strline													:	WSTRING(MAX_STRING_LENGTH);
END_VAR             										
VAR       
	lenght,pos												:	INT;          	
	tmp														:	WSTRING(MAX_STRING_LENGTH);
END_VAR

IF strline = ""
THEN
	cutWStrToSeperator										:= strline;
ELSE
	pos 													:= WFIND (strline,seperator);
	IF pos > 0 
	THEN
		cutWStrToSeperator									:= WLEFT(strline,pos-1);	
		Lenght												:= WLEN(strline);	
		IF Lenght > pos 
		THEN //write back string without seperator		
			tmp												:= WRIGHT(strline, Lenght - (pos - 1 + WLEN(seperator))); //Save rest
			MEMSET(ADR(strline), 0, TO_UDINT(Lenght) * 2);//delete complete string
			MEMCPY(ADR(strline), ADR(tmp), TO_UDINT(WLEN(tmp) * 2));
		ELSE //Delete stringline because seperator is at the end
			MEMSET(ADR(strline), 0, TO_UDINT(Lenght) * 2);//delete complete string
		END_IF              								
	ELSE                    								
		cutWStrToSeperator									:="";
	END_IF
END_IF

END_FUNCTION

